	__SYSTEM.TYPE_CLASS.TYPE_ULINT:
	
	convertResult := TryConvert_TOD_TO_ULINT(in, _ULINT);
	IF convertResult THEN
		convertAddress := ADR(_ULINT);
	END_IF
	
	__SYSTEM.TYPE_CLASS.TYPE_REAL:
	
	convertResult := TryConvert_TOD_TO_REAL(in, _REAL);
	IF convertResult THEN
		convertAddress := ADR(_REAL);
	END_IF
	
	__SYSTEM.TYPE_CLASS.TYPE_LREAL:
	
	convertResult := TryConvert_TOD_TO_LREAL(in, _LREAL);
	IF convertResult THEN
		convertAddress := ADR(_LREAL);
	END_IF
	
	__SYSTEM.TYPE_CLASS.TYPE_TIME:
	
	convertResult := TryConvert_TOD_TO_TIME(in, _TIME);
	IF convertResult THEN
		convertAddress := ADR(_TIME);
	END_IF
	
	__SYSTEM.TYPE_CLASS.TYPE_TIMEOFDAY:
	
	convertResult := TryConvert_TOD_TO_TOD(in, _TOD);
	IF convertResult THEN
		convertAddress := ADR(_TOD);
	END_IF
	
	__SYSTEM.TYPE_CLASS.TYPE_DATE:
	
	convertResult := TryConvert_TOD_TO_DATE(in, _DATE);
	IF convertResult THEN
		convertAddress := ADR(_DATE);
	END_IF
	
	__SYSTEM.TYPE_CLASS.TYPE_DATEANDTIME:
	
	convertResult := TryConvert_TOD_TO_DT(in, _DT);
	IF convertResult THEN
		convertAddress := ADR(_DT);
	END_IF
	
	__SYSTEM.TYPE_CLASS.TYPE_STRING:
	
	convertResult := TryConvert_TOD_TO_STRING(in, _STRING);
	IF convertResult THEN
		convertAddress := ADR(_STRING);
	END_IF
	
END_CASE

IF convertResult THEN
	memcpy(out.pValue,convertAddress,DINT_TO_UDINT(out.diSize));
END_IF

TryConvert_TOD_TO_Destination := convertResult;

END_FUNCTION

// ---- mobject-datatypes/Primitive/_DT.TcPOU
{attribute 'linkalways'} 
{attribute 'no_explicit_call' := 'This FB is a CLASS and must be accessed using methods or properties'}
{attribute 'enable_dynamic_creation'}
FUNCTION_BLOCK _DT EXTENDS DatatypeBase implements I_DT
VAR
	localData : DT;
	activeData : REFERENCE TO DT REF= localData;
END_VAR

PROPERTY PUBLIC Address : PVOID
GET
Address := ADR(activeData);
END_GET
END_PROPERTY

METHOD PUBLIC ClearReference
VAR_INPUT
END_VAR
activeData REF= localData;
END_METHOD

METHOD PUBLIC Clone : I_Datatype
VAR
    pClone : POINTER TO _DT;
END_VAR
pClone := __NEW(_DT(InitialValue := Value));
Clone := pClone^;
END_METHOD

METHOD FB_init : BOOL
VAR_INPUT
	bInitRetains : BOOL; // if TRUE, the retain variables are initialized (warm start / cold start)
	bInCopyCode : BOOL;  // if TRUE, the instance afterwards gets moved WORDo the copy code (online change)
	InitialValue : DT;
END_VAR
localData := InitialValue;
END_METHOD

METHOD PUBLIC MakeReferenceTo
VAR_INPUT
	ReferenceTarget : REFERENCE TO DT;
END_VAR
activeData REF= ReferenceTarget;
END_METHOD

METHOD PUBLIC SerializeWith
VAR_INPUT
	Serializer : I_Serializer;
END_VAR
Serializer.AddDateTime(activeData);
END_METHOD

PROPERTY PUBLIC Size : UDINT
GET
Size := SIZEOF(activeData);
END_GET
END_PROPERTY

METHOD PUBLIC TryConvertTo : BOOL
VAR_INPUT
	Destination : ANY;
END_VAR
TryConvertTo := TryConvert_DT_To_Destination(activeData, Destination);
END_METHOD

METHOD PUBLIC TryConvertTo_ : BOOL
VAR_INPUT
	Destination : I_Datatype;
END_VAR
VAR
	resultofBitConversion : BOOL;
	destinationAs_BIT : I_BIT;
	destinationAs_BOOL : I_BOOL;
	destinationAs_BYTE : I_BYTE;
	destinationAs_DINT : I_DINT;
	destinationAs_DT : I_DT;
	destinationAs_DWORD : I_DWORD;
	destinationAs_INT : I_INT;
	destinationAs_LINT : I_LINT;
	destinationAs_LREAL : I_LREAL;
	destinationAs_LWORD : I_LWORD;
	destinationAs_REAL : I_REAL;
	destinationAs_SINT : I_SINT;
	destinationAs_STRING : I_STRING;
	destinationAs_TOD : I_TOD;
	destinationAs_UDINT : I_UDINT;
	destinationAs_UINT : I_UINT;
	destinationAs_ULINT : I_ULINT;
	destinationAs_USINT : I_USINT;
	destinationAs_WORD : I_WORD;
END_VAR
IF destination.TryResolveAs_BIT(destinationAs_BIT) AND_THEN TryConvert_DT_TO_BOOL(activeData, resultofBitConversion) THEN
	destinationAs_BIT.Value := resultOfBitConversion;
	TryConvertTo_ := TRUE;
	RETURN;
END_IF

IF destination.TryResolveAs_BOOL(destinationAs_BOOL) THEN
	TryConvertTo_ := TryConvert_DT_TO_BOOL(activeData, destinationAs_BOOL.Value);
	RETURN;
END_IF
		
IF destination.TryResolveAs_BYTE(destinationAs_BYTE) THEN
	TryConvertTo_ := TryConvert_DT_TO_BYTE(activeData, destinationAs_BYTE.Value);
	RETURN;
END_IF

IF destination.TryResolveAs_DINT(destinationAs_DINT) THEN
	TryConvertTo_ := TryConvert_DT_TO_DINT(activeData, destinationAs_DINT.Value);
	RETURN;
END_IF

IF destination.TryResolveAs_DT(destinationAs_DT) THEN
	TryConvertTo_ := TryConvert_DT_TO_DT(activeData, destinationAs_DT.Value);
	RETURN;
END_IF

IF destination.TryResolveAs_DWORD(destinationAs_DWORD) THEN
	TryConvertTo_ := TryConvert_DT_TO_DWORD(activeData, destinationAs_DWORD.Value);
	RETURN;
END_IF

IF destination.TryResolveAs_INT(destinationAs_INT) THEN
	TryConvertTo_ := TryConvert_DT_TO_INT(activeData, destinationAs_INT.Value);
	RETURN;
END_IF

IF destination.TryResolveAs_LINT(destinationAs_LINT) THEN
	TryConvertTo_ := TryConvert_DT_TO_LINT(activeData, destinationAs_LINT.Value);
	RETURN;
END_IF

IF destination.TryResolveAs_LREAL(destinationAs_LREAL) THEN
	TryConvertTo_ := TryConvert_DT_TO_LREAL(activeData, destinationAs_LREAL.Value);
	RETURN;
END_IF

IF destination.TryResolveAs_LWORD(destinationAs_LWORD) THEN
	TryConvertTo_ := TryConvert_DT_TO_LWORD(activeData, destinationAs_LWORD.Value);
	RETURN;
END_IF

IF destination.TryResolveAs_REAL(destinationAs_REAL) THEN
	TryConvertTo_ := TryConvert_DT_TO_REAL(activeData, destinationAs_REAL.Value);
	RETURN;
END_IF

IF destination.TryResolveAs_SINT(destinationAs_SINT) THEN
	TryConvertTo_ := TryConvert_DT_TO_SINT(activeData, destinationAs_SINT.Value);
	RETURN;
END_IF

IF destination.TryResolveAs_STRING(destinationAs_STRING) THEN
	TryConvertTo_ := TryConvert_DT_TO_STRING(activeData, destinationAs_STRING.Value);
	RETURN;
END_IF

IF destination.TryResolveAs_TOD(destinationAs_TOD) THEN
	TryConvertTo_ := TryConvert_DT_TO_TOD(activeData, destinationAs_TOD.Value);
	RETURN;
END_IF

IF destination.TryResolveAs_UDINT(destinationAs_UDINT) THEN
	TryConvertTo_ := TryConvert_DT_TO_UDINT(activeData, destinationAs_UDINT.Value);
	RETURN;
END_IF

IF destination.TryResolveAs_UINT(destinationAs_UINT) THEN
	TryConvertTo_ := TryConvert_DT_TO_UINT(activeData, destinationAs_UINT.Value);
	RETURN;
END_IF

IF destination.TryResolveAs_ULINT(destinationAs_ULINT) THEN
	TryConvertTo_ := TryConvert_DT_TO_ULINT(activeData, destinationAs_ULINT.Value);
	RETURN;
END_IF

IF destination.TryResolveAs_USINT(destinationAs_USINT) THEN
	TryConvertTo_ := TryConvert_DT_TO_USINT(activeData, destinationAs_USINT.Value);
	RETURN;
END_IF

IF destination.TryResolveAs_WORD(destinationAs_WORD) THEN
	TryConvertTo_ := TryConvert_DT_TO_WORD(activeData, destinationAs_WORD.Value);
	RETURN;
END_IF
END_METHOD

METHOD TryDeserializeFrom : BOOL
VAR_INPUT
	Deserializer : I_Deserializer;
	Feedback : I_DeserializerFeedback;
END_VAR
TryDeserializeFrom := Deserializer.TryGetDateTime(activeData, Feedback);
END_METHOD

METHOD TryMakeReferenceTo : BOOL
VAR_INPUT
	Target : I_Datatype;
END_VAR
VAR
	pTargetData : POINTER TO DT;
END_VAR
IF NOT IsEquivalentTo(Target) THEN
	RETURN;
END_IF

pTargetData := Target.Address;
activeData REF= pTargetData^;
TryMakeReferenceTo := TRUE;
END_METHOD

METHOD PUBLIC TryResolveAs_DT : BOOL
VAR_INPUT
	Destination : REFERENCE TO I_DT;
END_VAR
Destination := THIS^;
TryResolveAs_DT := TRUE;
END_METHOD

PROPERTY PUBLIC TypeName : T_MAXSTRING
GET
TypeName := 'DT';
END_GET
END_PROPERTY

{warning disable C5410}
PROPERTY PUBLIC Value : REFERENCE TO DT
{warning restore C5410}
GET
Value REF= activeData;
END_GET
END_PROPERTY

END_FUNCTION_BLOCK

// ---- mobject-converters/Converters/DT_TO_/TryConvert_DT_TO_BOOL.TcPOU
FUNCTION TryConvert_DT_TO_BOOL : BOOL
VAR_INPUT
	in : DT;
	out : REFERENCE TO BOOL;
END_VAR

out := DT_TO_BOOL(in);
TryConvert_DT_TO_BOOL := TRUE;

END_FUNCTION

// ---- mobject-converters/Converters/DT_TO_/TryConvert_DT_TO_BYTE.TcPOU
FUNCTION TryConvert_DT_TO_BYTE : BOOL
VAR_INPUT
	in : DT;
	out : REFERENCE TO BYTE;
END_VAR

IF in > DatatypeLimits.MAX_VALUE_OF_DT_WHICH_CAN_BE_HELD_IN_A_BYTE THEN
	RETURN;
END_IF

out := DT_TO_BYTE(in);
TryConvert_DT_TO_BYTE := TRUE;

END_FUNCTION

// ---- mobject-converters/Converters/DT_TO_/TryConvert_DT_TO_DINT.TcPOU
FUNCTION TryConvert_DT_TO_DINT : BOOL
VAR_INPUT
	in : DT;
	out : REFERENCE TO DINT;
END_VAR

IF in > DatatypeLimits.MAX_VALUE_OF_DT_WHICH_CAN_BE_HELD_IN_A_DINT THEN
	RETURN;
END_IF

out := DT_TO_DINT(in);
TryConvert_DT_TO_DINT := TRUE;

END_FUNCTION

// ---- mobject-converters/Converters/DT_TO_/TryConvert_DT_TO_DT.TcPOU
FUNCTION TryConvert_DT_TO_DT : BOOL
VAR_INPUT
	in : DT;
	out : REFERENCE TO DT;
END_VAR

out := in;
TryConvert_DT_TO_DT := TRUE;

END_FUNCTION

// ---- mobject-converters/Converters/DT_TO_/TryConvert_DT_TO_DWORD.TcPOU
FUNCTION TryConvert_DT_TO_DWORD : BOOL
VAR_INPUT
	in : DT;
	out : REFERENCE TO DWORD;
END_VAR

out := DT_TO_DWORD(in);
TryConvert_DT_TO_DWORD := TRUE;

END_FUNCTION

// ---- mobject-converters/Converters/DT_TO_/TryConvert_DT_TO_LINT.TcPOU
FUNCTION TryConvert_DT_TO_LINT : BOOL
VAR_INPUT
	in : DT;
	out : REFERENCE TO LINT;
END_VAR

out := DT_TO_LINT(in);
TryConvert_DT_TO_LINT := TRUE;

END_FUNCTION

// ---- mobject-converters/Converters/DT_TO_/TryConvert_DT_TO_LWORD.TcPOU
FUNCTION TryConvert_DT_TO_LWORD : BOOL
VAR_INPUT
	in : DT;
	out : REFERENCE TO LWORD;
END_VAR

out := DT_TO_LWORD(in);
TryConvert_DT_TO_LWORD := TRUE;

END_FUNCTION

// ---- mobject-converters/Converters/DT_TO_/TryConvert_DT_TO_REAL.TcPOU
FUNCTION TryConvert_DT_TO_REAL : BOOL
VAR_INPUT
	in : DT;
	out : REFERENCE TO REAL;
END_VAR

out := DT_TO_REAL(in);
TryConvert_DT_TO_REAL := TRUE;

END_FUNCTION

// ---- mobject-converters/Converters/DT_TO_/TryConvert_DT_TO_TOD.TcPOU
FUNCTION TryConvert_DT_TO_TOD : BOOL
VAR_INPUT
	in : DT;
	out : REFERENCE TO TOD;
END_VAR

IF in > DatatypeLimits.MAX_VALUE_OF_DT_WHICH_CAN_BE_HELD_IN_A_TOD THEN
	RETURN;
END_IF

out := DT_TO_TOD(in);
TryConvert_DT_TO_TOD := TRUE;

END_FUNCTION

// ---- mobject-converters/Converters/DT_TO_/TryConvert_DT_TO_UINT.TcPOU
FUNCTION TryConvert_DT_TO_UINT : BOOL
VAR_INPUT
	in : DT;
	out : REFERENCE TO UINT;
END_VAR

IF in > DatatypeLimits.MAX_VALUE_OF_DT_WHICH_CAN_BE_HELD_IN_A_UINT THEN
	RETURN;
END_IF

out := DT_TO_UINT(in);
TryConvert_DT_TO_UINT := TRUE;

END_FUNCTION

// ---- mobject-converters/Converters/DT_TO_/TryConvert_DT_TO_ULINT.TcPOU
FUNCTION TryConvert_DT_TO_ULINT : BOOL
VAR_INPUT
	in : DT;
	out : REFERENCE TO ULINT;
END_VAR

out := DT_TO_ULINT(in);
TryConvert_DT_TO_ULINT := TRUE;

END_FUNCTION

// ---- mobject-datatypes/Primitive/_STRING.TcPOU
{attribute 'linkalways'} 
{attribute 'no_explicit_call' := 'This FB is a CLASS and must be accessed using methods or properties'}
{attribute 'enable_dynamic_creation'}
FUNCTION_BLOCK _STRING EXTENDS DatatypeBase implements I_STRING
VAR
	localData : T_MaxString;
	activeData : REFERENCE TO T_MaxString REF= localData;
END_VAR

PROPERTY PUBLIC Address : PVOID
GET
Address := ADR(activeData);
END_GET
END_PROPERTY

METHOD PUBLIC ClearReference
VAR_INPUT
END_VAR
activeData REF= localData;
END_METHOD

METHOD PUBLIC Clone : I_Datatype
VAR
    pClone : POINTER TO _STRING;
END_VAR
pClone := __NEW(_STRING(InitialValue := Value));
Clone := pClone^;
END_METHOD

METHOD FB_init : BOOL
VAR_INPUT
	bInitRetains : BOOL; // if TRUE, the retain variables are initialized (warm start / cold start)
	bInCopyCode : BOOL;  // if TRUE, the instance afterwards gets moved WORDo the copy code (online change)
	InitialValue : T_MaxString;
END_VAR
localData := InitialValue;
END_METHOD

PROPERTY PUBLIC Length : INT
GET
Length := len(activeData);
END_GET
END_PROPERTY

METHOD PUBLIC MakeReferenceTo
VAR_INPUT
	ReferenceTarget : REFERENCE TO T_MaxString;
END_VAR
activeData REF= ReferenceTarget;
END_METHOD

METHOD PUBLIC SerializeWith
VAR_INPUT
	Serializer : I_Serializer;
END_VAR
Serializer.AddString(activeData);
END_METHOD

PROPERTY PUBLIC Size : UDINT
GET
Size := SIZEOF(activeData);
END_GET
END_PROPERTY

METHOD PUBLIC TryConvertTo : BOOL
VAR_INPUT
	Destination : ANY;
END_VAR
TryConvertTo := TryConvert_STRING_TO_Destination(activeData, Destination);
END_METHOD

METHOD PUBLIC TryConvertTo_ : BOOL
VAR_INPUT
	Destination : I_Datatype;
END_VAR
VAR
	resultofBitConversion : BOOL;
	destinationAs_BIT : I_BIT;
	destinationAs_BOOL : I_BOOL;
	destinationAs_BYTE : I_BYTE;
	destinationAs_DINT : I_DINT;
	destinationAs_DT : I_DT;
	destinationAs_DWORD : I_DWORD;
	destinationAs_INT : I_INT;
	destinationAs_LINT : I_LINT;
	destinationAs_LREAL : I_LREAL;
	destinationAs_LWORD : I_LWORD;
	destinationAs_REAL : I_REAL;
	destinationAs_SINT : I_SINT;
	destinationAs_STRING : I_STRING;
	destinationAs_TOD : I_TOD;
	destinationAs_UDINT : I_UDINT;
	destinationAs_UINT : I_UINT;
	destinationAs_ULINT : I_ULINT;
	destinationAs_USINT : I_USINT;
	destinationAs_WORD : I_WORD;
END_VAR
IF destination.TryResolveAs_BIT(destinationAs_BIT) AND_THEN TryConvert_STRING_TO_BOOL(activeData, resultofBitConversion) THEN
	destinationAs_BIT.Value := resultOfBitConversion;
	TryConvertTo_ := TRUE;
	RETURN;
END_IF

IF destination.TryResolveAs_BOOL(destinationAs_BOOL) THEN
	TryConvertTo_ := TryConvert_STRING_TO_BOOL(activeData, destinationAs_BOOL.Value);
	RETURN;
END_IF
		
IF destination.TryResolveAs_BYTE(destinationAs_BYTE) THEN
	TryConvertTo_ := TryConvert_STRING_TO_BYTE(activeData, destinationAs_BYTE.Value);
	RETURN;
END_IF

IF destination.TryResolveAs_DINT(destinationAs_DINT) THEN
	TryConvertTo_ := TryConvert_STRING_TO_DINT(activeData, destinationAs_DINT.Value);
	RETURN;
END_IF

IF destination.TryResolveAs_DT(destinationAs_DT) THEN
	TryConvertTo_ := TryConvert_STRING_TO_DT(activeData, destinationAs_DT.Value);
	RETURN;
END_IF

IF destination.TryResolveAs_DWORD(destinationAs_DWORD) THEN
	TryConvertTo_ := TryConvert_STRING_TO_DWORD(activeData, destinationAs_DWORD.Value);
	RETURN;
END_IF

IF destination.TryResolveAs_INT(destinationAs_INT) THEN
	TryConvertTo_ := TryConvert_STRING_TO_INT(activeData, destinationAs_INT.Value);
	RETURN;
END_IF

IF destination.TryResolveAs_LINT(destinationAs_LINT) THEN
	TryConvertTo_ := TryConvert_STRING_TO_LINT(activeData, destinationAs_LINT.Value);
	RETURN;
END_IF

IF destination.TryResolveAs_LREAL(destinationAs_LREAL) THEN
	TryConvertTo_ := TryConvert_STRING_TO_LREAL(activeData, destinationAs_LREAL.Value);
	RETURN;
END_IF

IF destination.TryResolveAs_LWORD(destinationAs_LWORD) THEN
	TryConvertTo_ := TryConvert_STRING_TO_LWORD(activeData, destinationAs_LWORD.Value);
	RETURN;
END_IF

IF destination.TryResolveAs_REAL(destinationAs_REAL) THEN
	TryConvertTo_ := TryConvert_STRING_TO_REAL(activeData, destinationAs_REAL.Value);
	RETURN;
END_IF

IF destination.TryResolveAs_SINT(destinationAs_SINT) THEN
	TryConvertTo_ := TryConvert_STRING_TO_SINT(activeData, destinationAs_SINT.Value);
	RETURN;
END_IF

IF destination.TryResolveAs_STRING(destinationAs_STRING) THEN
	TryConvertTo_ := TryConvert_STRING_TO_STRING(activeData, destinationAs_STRING.Value);
	RETURN;
END_IF

IF destination.TryResolveAs_TOD(destinationAs_TOD) THEN
	TryConvertTo_ := TryConvert_STRING_TO_TOD(activeData, destinationAs_TOD.Value);
	RETURN;
END_IF

IF destination.TryResolveAs_UDINT(destinationAs_UDINT) THEN
	TryConvertTo_ := TryConvert_STRING_TO_UDINT(activeData, destinationAs_UDINT.Value);
	RETURN;
END_IF

IF destination.TryResolveAs_UINT(destinationAs_UINT) THEN
	TryConvertTo_ := TryConvert_STRING_TO_UINT(activeData, destinationAs_UINT.Value);
	RETURN;
END_IF

IF destination.TryResolveAs_ULINT(destinationAs_ULINT) THEN
	TryConvertTo_ := TryConvert_STRING_TO_ULINT(activeData, destinationAs_ULINT.Value);
	RETURN;
END_IF

IF destination.TryResolveAs_USINT(destinationAs_USINT) THEN
	TryConvertTo_ := TryConvert_STRING_TO_USINT(activeData, destinationAs_USINT.Value);
	RETURN;
END_IF

IF destination.TryResolveAs_WORD(destinationAs_WORD) THEN
	TryConvertTo_ := TryConvert_STRING_TO_WORD(activeData, destinationAs_WORD.Value);
	RETURN;
END_IF
END_METHOD

METHOD TryDeserializeFrom : BOOL
VAR_INPUT
	Deserializer : I_Deserializer;
	Feedback : I_DeserializerFeedback;
END_VAR
TryDeserializeFrom := Deserializer.TryGetString(activeData, Feedback);
END_METHOD

METHOD TryMakeReferenceTo : BOOL
VAR_INPUT
	Target : I_Datatype;
END_VAR
VAR
	pTargetData : POINTER TO T_MaxString;
END_VAR
IF NOT IsEquivalentTo(Target) THEN
	RETURN;
END_IF

pTargetData := Target.Address;
activeData REF= pTargetData^;
TryMakeReferenceTo := TRUE;
END_METHOD

METHOD PUBLIC TryResolveAs_STRING : BOOL
VAR_INPUT
	Destination : REFERENCE TO I_STRING;
END_VAR
Destination := THIS^;
TryResolveAs_STRING := TRUE;
END_METHOD

PROPERTY PUBLIC TypeName : T_MAXSTRING
GET
TypeName := 'STRING';
END_GET
END_PROPERTY

{warning disable C5410}
PROPERTY PUBLIC Value : REFERENCE TO T_MaxString
{warning restore C5410}
GET
Value REF= activeData;
END_GET
END_PROPERTY

END_FUNCTION_BLOCK

// ---- mobject-converters/Converters/STRING_TO_/TryConvert_STRING_TO_Destination.TcPOU
FUNCTION TryConvert_STRING_TO_Destination : BOOL
VAR_INPUT
	in : STRING;
	out : ANY;
END_VAR
VAR
	convertResult : BOOL := FALSE;
	convertAddress : PVOID;
	_BOOL : BOOL;
	_BYTE : BYTE;
	_WORD : WORD;
	_DWORD : DWORD;
	_LWORD : LWORD;
	_SINT : SINT;
	_INT : INT;
	_DINT : DINT;
	_LINT : LINT;
	_USINT : USINT;
	_UINT : UINT;
	_UDINT : UDINT;
	_ULINT : ULINT;
	_REAL : REAL;
	_LREAL : LREAL;
	_TIME : TIME;
	_TOD : TOD;
	_DATE : DATE;
	_DT : DT;
	_STRING : STRING;
END_VAR

CASE out.TypeClass OF
	__SYSTEM.TYPE_CLASS.TYPE_BOOL:
	
	convertResult := TryConvert_STRING_TO_BOOL(in, _BOOL);
	IF convertResult THEN
		convertAddress := ADR(_BOOL);
	END_IF
	
	__SYSTEM.TYPE_CLASS.TYPE_BYTE:
	
	convertResult := TryConvert_STRING_TO_BYTE(in, _BYTE);
	IF convertResult THEN
		convertAddress := ADR(_BYTE);
	END_IF
	
	__SYSTEM.TYPE_CLASS.TYPE_WORD:
	
	convertResult := TryConvert_STRING_TO_WORD(in, _WORD);
	IF convertResult THEN
		convertAddress := ADR(_WORD);
	END_IF
	
	__SYSTEM.TYPE_CLASS.TYPE_DWORD:
	
	convertResult := TryConvert_STRING_TO_DWORD(in, _DWORD);
	IF convertResult THEN
		convertAddress := ADR(_DWORD);
	END_IF
	
	__SYSTEM.TYPE_CLASS.TYPE_LWORD:
	
	convertResult := TryConvert_STRING_TO_LWORD(in, _LWORD);
	IF convertResult THEN
		convertAddress := ADR(_LWORD);
	END_IF
	
	__SYSTEM.TYPE_CLASS.TYPE_SINT:
	
	convertResult := TryConvert_STRING_TO_SINT(in, _SINT);
	IF convertResult THEN
		convertAddress := ADR(_SINT);
	END_IF
	
	__SYSTEM.TYPE_CLASS.TYPE_INT:
	
	convertResult := TryConvert_STRING_TO_INT(in, _INT);
	IF convertResult THEN
		convertAddress := ADR(_INT);
	END_IF
	
	__SYSTEM.TYPE_CLASS.TYPE_DINT:
	
	convertResult := TryConvert_STRING_TO_DINT(in, _DINT);
	IF convertResult THEN
		convertAddress := ADR(_DINT);
	END_IF
	
	__SYSTEM.TYPE_CLASS.TYPE_LINT:
	
	convertResult := TryConvert_STRING_TO_LINT(in, _LINT);
	IF convertResult THEN
		convertAddress := ADR(_LINT);
	END_IF
	
	__SYSTEM.TYPE_CLASS.TYPE_USINT:
	
	convertResult := TryConvert_STRING_TO_USINT(in, _USINT);
	IF convertResult THEN
		convertAddress := ADR(_USINT);
	END_IF
	
	__SYSTEM.TYPE_CLASS.TYPE_UINT:
	
	convertResult := TryConvert_STRING_TO_UINT(in, _UINT);
	IF convertResult THEN
		convertAddress := ADR(_UINT);
	END_IF
	
	__SYSTEM.TYPE_CLASS.TYPE_UDINT:
	
	convertResult := TryConvert_STRING_TO_UDINT(in, _UDINT);
	IF convertResult THEN
		convertAddress := ADR(_UDINT);
	END_IF
	
	__SYSTEM.TYPE_CLASS.TYPE_ULINT:
	
	convertResult := TryConvert_STRING_TO_ULINT(in, _ULINT);
	IF convertResult THEN
		convertAddress := ADR(_ULINT);
	END_IF
	
	__SYSTEM.TYPE_CLASS.TYPE_REAL:
	
	convertResult := TryConvert_STRING_TO_REAL(in, _REAL);
	IF convertResult THEN
		convertAddress := ADR(_REAL);
	END_IF
	
	__SYSTEM.TYPE_CLASS.TYPE_LREAL:
	
	convertResult := TryConvert_STRING_TO_LREAL(in, _LREAL);
	IF convertResult THEN
		convertAddress := ADR(_LREAL);
	END_IF
	
	__SYSTEM.TYPE_CLASS.TYPE_TIME:
	
	convertResult := TryConvert_STRING_TO_TIME(in, _TIME);
	IF convertResult THEN
		convertAddress := ADR(_TIME);
	END_IF
	
	__SYSTEM.TYPE_CLASS.TYPE_TIMEOFDAY:
	
	convertResult := TryConvert_STRING_TO_TOD(in, _TOD);
	IF convertResult THEN
		convertAddress := ADR(_TOD);
	END_IF
	
	__SYSTEM.TYPE_CLASS.TYPE_DATE:
	
	convertResult := TryConvert_STRING_TO_DATE(in, _DATE);
	IF convertResult THEN
		convertAddress := ADR(_DATE);
	END_IF
	
	__SYSTEM.TYPE_CLASS.TYPE_DATEANDTIME:
	
	convertResult := TryConvert_STRING_TO_DT(in, _DT);
	IF convertResult THEN
		convertAddress := ADR(_DT);
	END_IF
	
	__SYSTEM.TYPE_CLASS.TYPE_STRING:
	
	convertResult := TryConvert_STRING_TO_STRING(in, _STRING);
	IF convertResult THEN
		convertAddress := ADR(_STRING);
	END_IF
	
END_CASE

IF convertResult THEN
	memcpy(out.pValue,convertAddress,DINT_TO_UDINT(out.diSize));
END_IF

TryConvert_STRING_TO_Destination := convertResult;

END_FUNCTION

// ---- mobject-converters/Converters/STRING_TO_/TryConvert_STRING_TO_BYTE.TcPOU
FUNCTION TryConvert_STRING_TO_BYTE : BOOL
VAR_INPUT
	in : STRING;
	out : REFERENCE TO BYTE;
END_VAR

IF in <> BYTE_TO_STRING(STRING_TO_BYTE(in)) THEN
	RETURN;
END_IF

out := STRING_TO_BYTE(in);
TryConvert_STRING_TO_BYTE := TRUE;

END_FUNCTION

// ---- mobject-converters/Converters/STRING_TO_/TryConvert_STRING_TO_WORD.TcPOU
FUNCTION TryConvert_STRING_TO_WORD : BOOL
VAR_INPUT
	in : STRING;
	out : REFERENCE TO WORD;
END_VAR

IF in <> WORD_TO_STRING(STRING_TO_WORD(in)) THEN
	RETURN;
END_IF

out := STRING_TO_WORD(in);
TryConvert_STRING_TO_WORD := TRUE;

END_FUNCTION

// ---- mobject-converters/Converters/STRING_TO_/TryConvert_STRING_TO_DWORD.TcPOU
FUNCTION TryConvert_STRING_TO_DWORD : BOOL
VAR_INPUT
	in : STRING;
	out : REFERENCE TO DWORD;
END_VAR

IF in <> DWORD_TO_STRING(STRING_TO_DWORD(in)) THEN
	RETURN;
END_IF

out := STRING_TO_DWORD(in);
TryConvert_STRING_TO_DWORD := TRUE;

END_FUNCTION

// ---- mobject-converters/Converters/STRING_TO_/TryConvert_STRING_TO_SINT.TcPOU
FUNCTION TryConvert_STRING_TO_SINT : BOOL
VAR_INPUT
	in : STRING;
	out : REFERENCE TO SINT;
END_VAR

IF in <> SINT_TO_STRING(STRING_TO_SINT(in)) THEN
	RETURN;
END_IF

out := STRING_TO_SINT(in);
TryConvert_STRING_TO_SINT := TRUE;

END_FUNCTION

// ---- mobject-converters/Converters/STRING_TO_/TryConvert_STRING_TO_DINT.TcPOU
FUNCTION TryConvert_STRING_TO_DINT : BOOL
VAR_INPUT
	in : STRING;
	out : REFERENCE TO DINT;
END_VAR

IF in <> DINT_TO_STRING(STRING_TO_DINT(in)) THEN
	RETURN;
END_IF

out := STRING_TO_DINT(in);
TryConvert_STRING_TO_DINT := TRUE;

END_FUNCTION

// ---- mobject-converters/Converters/STRING_TO_/TryConvert_STRING_TO_USINT.TcPOU
FUNCTION TryConvert_STRING_TO_USINT : BOOL
VAR_INPUT
	in : STRING;
	out : REFERENCE TO USINT;
END_VAR

IF in <> USINT_TO_STRING(STRING_TO_USINT(in)) THEN
	RETURN;
END_IF

out := STRING_TO_USINT(in);
TryConvert_STRING_TO_USINT := TRUE;

END_FUNCTION

// ---- mobject-converters/Converters/STRING_TO_/TryConvert_STRING_TO_UINT.TcPOU
FUNCTION TryConvert_STRING_TO_UINT : BOOL
VAR_INPUT
	in : STRING;
	out : REFERENCE TO UINT;
END_VAR

IF in <> UINT_TO_STRING(STRING_TO_UINT(in)) THEN
	RETURN;
END_IF

out := STRING_TO_UINT(in);
TryConvert_STRING_TO_UINT := TRUE;

END_FUNCTION

// ---- mobject-converters/Converters/STRING_TO_/TryConvert_STRING_TO_ULINT.TcPOU
FUNCTION TryConvert_STRING_TO_ULINT : BOOL
VAR_INPUT
	in : STRING;
	out : REFERENCE TO ULINT;
END_VAR

IF in <> ULINT_TO_STRING(STRING_TO_ULINT(in)) THEN
	RETURN;
END_IF

out := STRING_TO_ULINT(in);
TryConvert_STRING_TO_ULINT := TRUE;

END_FUNCTION

// ---- mobject-converters/Converters/STRING_TO_/TryConvert_STRING_TO_REAL.TcPOU
FUNCTION TryConvert_STRING_TO_REAL : BOOL
VAR_INPUT
	in : STRING;
	out : REFERENCE TO REAL;
END_VAR

IF in <> REAL_TO_STRING(STRING_TO_REAL(in)) THEN
	RETURN;
END_IF

out := STRING_TO_REAL(in);
TryConvert_STRING_TO_REAL := TRUE;

END_FUNCTION

// ---- mobject-converters/Converters/STRING_TO_/TryConvert_STRING_TO_LREAL.TcPOU
FUNCTION TryConvert_STRING_TO_LREAL : BOOL
VAR_INPUT
	in : STRING;
	out : REFERENCE TO LREAL;
END_VAR

IF in <> LREAL_TO_STRING(STRING_TO_LREAL(in)) THEN
	RETURN;
END_IF

out := STRING_TO_LREAL(in);
TryConvert_STRING_TO_LREAL := TRUE;

END_FUNCTION

// ---- mobject-converters/Converters/STRING_TO_/TryConvert_STRING_TO_TOD.TcPOU
FUNCTION TryConvert_STRING_TO_TOD : BOOL
VAR_INPUT
	in : STRING;
	out : REFERENCE TO TOD;
END_VAR

IF in <> TOD_TO_STRING(STRING_TO_TOD(in)) THEN
	RETURN;
END_IF

out := STRING_TO_TOD(in);
TryConvert_STRING_TO_TOD := TRUE;

END_FUNCTION

// ---- mobject-converters/Converters/STRING_TO_/TryConvert_STRING_TO_DATE.TcPOU
FUNCTION TryConvert_STRING_TO_DATE : BOOL
VAR_INPUT
	in : STRING;
	out : REFERENCE TO DATE;
END_VAR

IF in <> DATE_TO_STRING(STRING_TO_DATE(in)) THEN
	RETURN;
END_IF

out := STRING_TO_DATE(in);
TryConvert_STRING_TO_DATE := TRUE;

END_FUNCTION

// ---- mobject-converters/Converters/STRING_TO_/TryConvert_STRING_TO_STRING.TcPOU
FUNCTION TryConvert_STRING_TO_STRING : BOOL
VAR_INPUT
	in : STRING;
	out : REFERENCE TO STRING;
END_VAR

out := in;
TryConvert_STRING_TO_STRING := TRUE;

END_FUNCTION

// ---- mobject-converters/Converters/TOD_TO_/TryConvert_TOD_TO_BOOL.TcPOU
FUNCTION TryConvert_TOD_TO_BOOL : BOOL
VAR_INPUT
	in : TOD;
	out : REFERENCE TO BOOL;
END_VAR

out := TOD_TO_BOOL(in);
TryConvert_TOD_TO_BOOL := TRUE;

END_FUNCTION

// ---- mobject-converters/Converters/TOD_TO_/TryConvert_TOD_TO_BYTE.TcPOU
FUNCTION TryConvert_TOD_TO_BYTE : BOOL
VAR_INPUT
	in : TOD;
	out : REFERENCE TO BYTE;
END_VAR

IF in > DatatypeLimits.MAX_VALUE_OF_TOD_WHICH_CAN_BE_HELD_IN_A_BYTE THEN
	RETURN;
END_IF

out := TOD_TO_BYTE(in);
TryConvert_TOD_TO_BYTE := TRUE;

END_FUNCTION

// ---- mobject-converters/Converters/TOD_TO_/TryConvert_TOD_TO_WORD.TcPOU
FUNCTION TryConvert_TOD_TO_WORD : BOOL
VAR_INPUT
	in : TOD;
	out : REFERENCE TO WORD;
END_VAR

IF in > DatatypeLimits.MAX_VALUE_OF_TOD_WHICH_CAN_BE_HELD_IN_A_WORD THEN
	RETURN;
END_IF

out := TOD_TO_WORD(in);
TryConvert_TOD_TO_WORD := TRUE;

END_FUNCTION

// ---- mobject-converters/Converters/TOD_TO_/TryConvert_TOD_TO_INT.TcPOU
FUNCTION TryConvert_TOD_TO_INT : BOOL
VAR_INPUT
	in : TOD;
	out : REFERENCE TO INT;
END_VAR

IF in > DatatypeLimits.MAX_VALUE_OF_TOD_WHICH_CAN_BE_HELD_IN_A_INT THEN
	RETURN;
END_IF

out := TOD_TO_INT(in);
TryConvert_TOD_TO_INT := TRUE;

END_FUNCTION

// ---- mobject-converters/Converters/TOD_TO_/TryConvert_TOD_TO_LINT.TcPOU
FUNCTION TryConvert_TOD_TO_LINT : BOOL
VAR_INPUT
	in : TOD;
	out : REFERENCE TO LINT;
END_VAR

out := TOD_TO_LINT(in);
TryConvert_TOD_TO_LINT := TRUE;

END_FUNCTION

// ---- mobject-converters/Converters/TOD_TO_/TryConvert_TOD_TO_USINT.TcPOU
FUNCTION TryConvert_TOD_TO_USINT : BOOL
VAR_INPUT
	in : TOD;
	out : REFERENCE TO USINT;
END_VAR

IF in > DatatypeLimits.MAX_VALUE_OF_TOD_WHICH_CAN_BE_HELD_IN_A_USINT THEN
	RETURN;
END_IF

out := TOD_TO_USINT(in);
TryConvert_TOD_TO_USINT := TRUE;

END_FUNCTION

// ---- mobject-converters/Converters/TOD_TO_/TryConvert_TOD_TO_REAL.TcPOU
FUNCTION TryConvert_TOD_TO_REAL : BOOL
VAR_INPUT
	in : TOD;
	out : REFERENCE TO REAL;
END_VAR

out := TOD_TO_REAL(in);
TryConvert_TOD_TO_REAL := TRUE;

END_FUNCTION

// ---- mobject-converters/Converters/TOD_TO_/TryConvert_TOD_TO_TIME.TcPOU
FUNCTION TryConvert_TOD_TO_TIME : BOOL
VAR_INPUT
	in : TOD;
	out : REFERENCE TO TIME;
END_VAR

out := TOD_TO_TIME(in);
TryConvert_TOD_TO_TIME := TRUE;

END_FUNCTION

// ---- mobject-converters/Converters/ULINT_TO_/TryConvert_ULINT_TO_BYTE.TcPOU
FUNCTION TryConvert_ULINT_TO_BYTE : BOOL
VAR_INPUT
	in : ULINT;
	out : REFERENCE TO BYTE;
END_VAR

IF in > DatatypeLimits.MAX_VALUE_OF_ULINT_WHICH_CAN_BE_HELD_IN_A_BYTE THEN
	RETURN;
END_IF

out := ULINT_TO_BYTE(in);
TryConvert_ULINT_TO_BYTE := TRUE;

END_FUNCTION

// ---- mobject-converters/Converters/ULINT_TO_/TryConvert_ULINT_TO_WORD.TcPOU
FUNCTION TryConvert_ULINT_TO_WORD : BOOL
VAR_INPUT
	in : ULINT;
	out : REFERENCE TO WORD;
END_VAR

IF in > DatatypeLimits.MAX_VALUE_OF_ULINT_WHICH_CAN_BE_HELD_IN_A_WORD THEN
	RETURN;
END_IF

out := ULINT_TO_WORD(in);
TryConvert_ULINT_TO_WORD := TRUE;

END_FUNCTION

// ---- mobject-converters/Converters/ULINT_TO_/TryConvert_ULINT_TO_DWORD.TcPOU
FUNCTION TryConvert_ULINT_TO_DWORD : BOOL
VAR_INPUT
	in : ULINT;
	out : REFERENCE TO DWORD;
END_VAR

IF in > DatatypeLimits.MAX_VALUE_OF_ULINT_WHICH_CAN_BE_HELD_IN_A_DWORD THEN
	RETURN;
END_IF

out := ULINT_TO_DWORD(in);
TryConvert_ULINT_TO_DWORD := TRUE;

END_FUNCTION

// ---- mobject-converters/Converters/ULINT_TO_/TryConvert_ULINT_TO_INT.TcPOU
FUNCTION TryConvert_ULINT_TO_INT : BOOL
VAR_INPUT
	in : ULINT;
	out : REFERENCE TO INT;
END_VAR

IF in > DatatypeLimits.MAX_VALUE_OF_ULINT_WHICH_CAN_BE_HELD_IN_A_INT THEN
	RETURN;
END_IF

out := ULINT_TO_INT(in);
TryConvert_ULINT_TO_INT := TRUE;

END_FUNCTION

// ---- mobject-converters/Converters/ULINT_TO_/TryConvert_ULINT_TO_LINT.TcPOU
FUNCTION TryConvert_ULINT_TO_LINT : BOOL
VAR_INPUT
	in : ULINT;
	out : REFERENCE TO LINT;
END_VAR

IF in > DatatypeLimits.MAX_VALUE_OF_ULINT_WHICH_CAN_BE_HELD_IN_A_LINT THEN
	RETURN;
END_IF

out := ULINT_TO_LINT(in);
TryConvert_ULINT_TO_LINT := TRUE;

END_FUNCTION

// ---- mobject-converters/Converters/ULINT_TO_/TryConvert_ULINT_TO_UINT.TcPOU
FUNCTION TryConvert_ULINT_TO_UINT : BOOL
VAR_INPUT
	in : ULINT;
	out : REFERENCE TO UINT;
END_VAR

IF in > DatatypeLimits.MAX_VALUE_OF_ULINT_WHICH_CAN_BE_HELD_IN_A_UINT THEN
	RETURN;
END_IF

out := ULINT_TO_UINT(in);
TryConvert_ULINT_TO_UINT := TRUE;

END_FUNCTION

// ---- mobject-converters/Converters/ULINT_TO_/TryConvert_ULINT_TO_ULINT.TcPOU
FUNCTION TryConvert_ULINT_TO_ULINT : BOOL
VAR_INPUT
	in : ULINT;
	out : REFERENCE TO ULINT;
END_VAR

out := in;
TryConvert_ULINT_TO_ULINT := TRUE;

END_FUNCTION

// ---- mobject-converters/Converters/ULINT_TO_/TryConvert_ULINT_TO_REAL.TcPOU
FUNCTION TryConvert_ULINT_TO_REAL : BOOL
VAR_INPUT
	in : ULINT;
	out : REFERENCE TO REAL;
END_VAR

out := ULINT_TO_REAL(in);
TryConvert_ULINT_TO_REAL := TRUE;

END_FUNCTION

// ---- mobject-converters/Converters/ULINT_TO_/TryConvert_ULINT_TO_LREAL.TcPOU
FUNCTION TryConvert_ULINT_TO_LREAL : BOOL
VAR_INPUT
	in : ULINT;
	out : REFERENCE TO LREAL;
END_VAR

out := ULINT_TO_LREAL(in);
TryConvert_ULINT_TO_LREAL := TRUE;

END_FUNCTION

// ---- mobject-converters/Converters/ULINT_TO_/TryConvert_ULINT_TO_TIME.TcPOU
FUNCTION TryConvert_ULINT_TO_TIME : BOOL
VAR_INPUT
	in : ULINT;
	out : REFERENCE TO TIME;
END_VAR

IF in > DatatypeLimits.MAX_VALUE_OF_ULINT_WHICH_CAN_BE_HELD_IN_A_TIME THEN
	RETURN;
END_IF

out := ULINT_TO_TIME(in);
TryConvert_ULINT_TO_TIME := TRUE;

END_FUNCTION

// ---- mobject-converters/Converters/ULINT_TO_/TryConvert_ULINT_TO_TOD.TcPOU
FUNCTION TryConvert_ULINT_TO_TOD : BOOL
VAR_INPUT
	in : ULINT;
	out : REFERENCE TO TOD;
END_VAR

IF in > DatatypeLimits.MAX_VALUE_OF_ULINT_WHICH_CAN_BE_HELD_IN_A_TOD THEN
	RETURN;
END_IF

out := ULINT_TO_TOD(in);
TryConvert_ULINT_TO_TOD := TRUE;

END_FUNCTION

// ---- mobject-converters/Converters/ULINT_TO_/TryConvert_ULINT_TO_DATE.TcPOU
FUNCTION TryConvert_ULINT_TO_DATE : BOOL
VAR_INPUT
	in : ULINT;
	out : REFERENCE TO DATE;
END_VAR

IF in > DatatypeLimits.MAX_VALUE_OF_ULINT_WHICH_CAN_BE_HELD_IN_A_DATE THEN
	RETURN;
END_IF

out := ULINT_TO_DATE(in);
TryConvert_ULINT_TO_DATE := TRUE;

END_FUNCTION

// ---- mobject-converters/Converters/UINT_TO_/TryConvert_UINT_TO_BOOL.TcPOU
FUNCTION TryConvert_UINT_TO_BOOL : BOOL
VAR_INPUT
	in : UINT;
	out : REFERENCE TO BOOL;
END_VAR

out := UINT_TO_BOOL(in);
TryConvert_UINT_TO_BOOL := TRUE;

END_FUNCTION

// ---- mobject-converters/Converters/UINT_TO_/TryConvert_UINT_TO_DWORD.TcPOU
FUNCTION TryConvert_UINT_TO_DWORD : BOOL
VAR_INPUT
	in : UINT;
	out : REFERENCE TO DWORD;
END_VAR

out := UINT_TO_DWORD(in);
TryConvert_UINT_TO_DWORD := TRUE;

END_FUNCTION

// ---- mobject-converters/Converters/UINT_TO_/TryConvert_UINT_TO_SINT.TcPOU
FUNCTION TryConvert_UINT_TO_SINT : BOOL
VAR_INPUT
	in : UINT;
	out : REFERENCE TO SINT;
END_VAR

IF in > DatatypeLimits.MAX_VALUE_OF_UINT_WHICH_CAN_BE_HELD_IN_A_SINT THEN
	RETURN;
END_IF

out := UINT_TO_SINT(in);
TryConvert_UINT_TO_SINT := TRUE;

END_FUNCTION

// ---- mobject-converters/Converters/UINT_TO_/TryConvert_UINT_TO_INT.TcPOU
FUNCTION TryConvert_UINT_TO_INT : BOOL
VAR_INPUT
	in : UINT;
	out : REFERENCE TO INT;
END_VAR

IF in > DatatypeLimits.MAX_VALUE_OF_UINT_WHICH_CAN_BE_HELD_IN_A_INT THEN
	RETURN;
END_IF

out := UINT_TO_INT(in);
TryConvert_UINT_TO_INT := TRUE;

END_FUNCTION

// ---- mobject-converters/Converters/UINT_TO_/TryConvert_UINT_TO_LINT.TcPOU
FUNCTION TryConvert_UINT_TO_LINT : BOOL
VAR_INPUT
	in : UINT;
	out : REFERENCE TO LINT;
END_VAR

out := UINT_TO_LINT(in);
TryConvert_UINT_TO_LINT := TRUE;

END_FUNCTION

// ---- mobject-converters/Converters/UINT_TO_/TryConvert_UINT_TO_UINT.TcPOU
FUNCTION TryConvert_UINT_TO_UINT : BOOL
VAR_INPUT
	in : UINT;
	out : REFERENCE TO UINT;
END_VAR

out := in;
TryConvert_UINT_TO_UINT := TRUE;

END_FUNCTION

// ---- mobject-converters/Converters/UINT_TO_/TryConvert_UINT_TO_UDINT.TcPOU
FUNCTION TryConvert_UINT_TO_UDINT : BOOL
VAR_INPUT
	in : UINT;
	out : REFERENCE TO UDINT;
END_VAR

out := UINT_TO_UDINT(in);
TryConvert_UINT_TO_UDINT := TRUE;

END_FUNCTION

// ---- mobject-converters/Converters/UINT_TO_/TryConvert_UINT_TO_REAL.TcPOU
FUNCTION TryConvert_UINT_TO_REAL : BOOL
VAR_INPUT
	in : UINT;
	out : REFERENCE TO REAL;
END_VAR

out := UINT_TO_REAL(in);
TryConvert_UINT_TO_REAL := TRUE;

END_FUNCTION

// ---- mobject-converters/Converters/UINT_TO_/TryConvert_UINT_TO_LREAL.TcPOU
FUNCTION TryConvert_UINT_TO_LREAL : BOOL
VAR_INPUT
	in : UINT;
	out : REFERENCE TO LREAL;
END_VAR

out := UINT_TO_LREAL(in);
TryConvert_UINT_TO_LREAL := TRUE;

END_FUNCTION

// ---- mobject-converters/Converters/UINT_TO_/TryConvert_UINT_TO_TIME.TcPOU
FUNCTION TryConvert_UINT_TO_TIME : BOOL
VAR_INPUT
	in : UINT;
	out : REFERENCE TO TIME;
END_VAR

out := UINT_TO_TIME(in);
TryConvert_UINT_TO_TIME := TRUE;

END_FUNCTION

// ---- mobject-converters/Converters/UINT_TO_/TryConvert_UINT_TO_TOD.TcPOU
FUNCTION TryConvert_UINT_TO_TOD : BOOL
VAR_INPUT
	in : UINT;
	out : REFERENCE TO TOD;
END_VAR

out := UINT_TO_TOD(in);
TryConvert_UINT_TO_TOD := TRUE;

END_FUNCTION

// ---- mobject-converters/Converters/UINT_TO_/TryConvert_UINT_TO_DATE.TcPOU
FUNCTION TryConvert_UINT_TO_DATE : BOOL
VAR_INPUT
	in : UINT;
	out : REFERENCE TO DATE;
END_VAR

out := UINT_TO_DATE(in);
TryConvert_UINT_TO_DATE := TRUE;

END_FUNCTION

// ---- mobject-converters/Converters/USINT_TO_/TryConvert_USINT_TO_WORD.TcPOU
FUNCTION TryConvert_USINT_TO_WORD : BOOL
VAR_INPUT
	in : USINT;
	out : REFERENCE TO WORD;
END_VAR

out := USINT_TO_WORD(in);
TryConvert_USINT_TO_WORD := TRUE;

END_FUNCTION

// ---- mobject-converters/Converters/USINT_TO_/TryConvert_USINT_TO_DWORD.TcPOU
FUNCTION TryConvert_USINT_TO_DWORD : BOOL
VAR_INPUT
	in : USINT;
	out : REFERENCE TO DWORD;
END_VAR

out := USINT_TO_DWORD(in);
TryConvert_USINT_TO_DWORD := TRUE;

END_FUNCTION

// ---- mobject-converters/Converters/USINT_TO_/TryConvert_USINT_TO_SINT.TcPOU
FUNCTION TryConvert_USINT_TO_SINT : BOOL
VAR_INPUT
	in : USINT;
	out : REFERENCE TO SINT;
END_VAR

IF in > DatatypeLimits.MAX_VALUE_OF_USINT_WHICH_CAN_BE_HELD_IN_A_SINT THEN
	RETURN;
END_IF

out := USINT_TO_SINT(in);
TryConvert_USINT_TO_SINT := TRUE;

END_FUNCTION

// ---- mobject-converters/Converters/USINT_TO_/TryConvert_USINT_TO_LINT.TcPOU
FUNCTION TryConvert_USINT_TO_LINT : BOOL
VAR_INPUT
	in : USINT;
	out : REFERENCE TO LINT;
END_VAR

out := USINT_TO_LINT(in);
TryConvert_USINT_TO_LINT := TRUE;

END_FUNCTION

// ---- mobject-converters/Converters/USINT_TO_/TryConvert_USINT_TO_USINT.TcPOU
FUNCTION TryConvert_USINT_TO_USINT : BOOL
VAR_INPUT
	in : USINT;
	out : REFERENCE TO USINT;
END_VAR

out := in;
TryConvert_USINT_TO_USINT := TRUE;

END_FUNCTION

// ---- mobject-converters/Converters/USINT_TO_/TryConvert_USINT_TO_UDINT.TcPOU
FUNCTION TryConvert_USINT_TO_UDINT : BOOL
VAR_INPUT
	in : USINT;
	out : REFERENCE TO UDINT;
END_VAR

out := USINT_TO_UDINT(in);
TryConvert_USINT_TO_UDINT := TRUE;

END_FUNCTION

// ---- mobject-converters/Converters/USINT_TO_/TryConvert_USINT_TO_REAL.TcPOU
FUNCTION TryConvert_USINT_TO_REAL : BOOL
VAR_INPUT
	in : USINT;
	out : REFERENCE TO REAL;
END_VAR

out := USINT_TO_REAL(in);
TryConvert_USINT_TO_REAL := TRUE;

END_FUNCTION

// ---- mobject-converters/Converters/USINT_TO_/TryConvert_USINT_TO_LREAL.TcPOU
FUNCTION TryConvert_USINT_TO_LREAL : BOOL
VAR_INPUT
	in : USINT;
	out : REFERENCE TO LREAL;
END_VAR

out := USINT_TO_LREAL(in);
TryConvert_USINT_TO_LREAL := TRUE;

END_FUNCTION

// ---- mobject-converters/Converters/USINT_TO_/TryConvert_USINT_TO_TIME.TcPOU
FUNCTION TryConvert_USINT_TO_TIME : BOOL
VAR_INPUT
	in : USINT;
	out : REFERENCE TO TIME;
END_VAR

out := USINT_TO_TIME(in);
TryConvert_USINT_TO_TIME := TRUE;

END_FUNCTION

// ---- mobject-converters/Converters/USINT_TO_/TryConvert_USINT_TO_DATE.TcPOU
FUNCTION TryConvert_USINT_TO_DATE : BOOL
VAR_INPUT
	in : USINT;
	out : REFERENCE TO DATE;
END_VAR

out := USINT_TO_DATE(in);
TryConvert_USINT_TO_DATE := TRUE;

END_FUNCTION

// ---- mobject-converters/Converters/USINT_TO_/TryConvert_USINT_TO_STRING.TcPOU
FUNCTION TryConvert_USINT_TO_STRING : BOOL
VAR_INPUT
	in : USINT;
	out : REFERENCE TO STRING;
END_VAR

out := USINT_TO_STRING(in);
TryConvert_USINT_TO_STRING := TRUE;

END_FUNCTION

// ---- mobject-converters/Converters/DWORD_TO_/TryConvert_DWORD_TO_BYTE.TcPOU
FUNCTION TryConvert_DWORD_TO_BYTE : BOOL
VAR_INPUT
	in : DWORD;
	out : REFERENCE TO BYTE;
END_VAR

IF in > DatatypeLimits.MAX_VALUE_OF_DWORD_WHICH_CAN_BE_HELD_IN_A_BYTE THEN
	RETURN;
END_IF

out := DWORD_TO_BYTE(in);
TryConvert_DWORD_TO_BYTE := TRUE;

END_FUNCTION

// ---- mobject-converters/Converters/DWORD_TO_/TryConvert_DWORD_TO_DWORD.TcPOU
FUNCTION TryConvert_DWORD_TO_DWORD : BOOL
VAR_INPUT
	in : DWORD;
	out : REFERENCE TO DWORD;
END_VAR

out := in;
TryConvert_DWORD_TO_DWORD := TRUE;

END_FUNCTION

// ---- mobject-converters/Converters/DWORD_TO_/TryConvert_DWORD_TO_LWORD.TcPOU
FUNCTION TryConvert_DWORD_TO_LWORD : BOOL
VAR_INPUT
	in : DWORD;
	out : REFERENCE TO LWORD;
END_VAR

out := DWORD_TO_LWORD(in);
TryConvert_DWORD_TO_LWORD := TRUE;

END_FUNCTION

// ---- mobject-converters/Converters/DWORD_TO_/TryConvert_DWORD_TO_INT.TcPOU
FUNCTION TryConvert_DWORD_TO_INT : BOOL
VAR_INPUT
	in : DWORD;
	out : REFERENCE TO INT;
END_VAR

IF in > DatatypeLimits.MAX_VALUE_OF_DWORD_WHICH_CAN_BE_HELD_IN_A_INT THEN
	RETURN;
END_IF

out := DWORD_TO_INT(in);
TryConvert_DWORD_TO_INT := TRUE;

END_FUNCTION

// ---- mobject-converters/Converters/DWORD_TO_/TryConvert_DWORD_TO_DINT.TcPOU
FUNCTION TryConvert_DWORD_TO_DINT : BOOL
VAR_INPUT
	in : DWORD;
	out : REFERENCE TO DINT;
END_VAR

IF in > DatatypeLimits.MAX_VALUE_OF_DWORD_WHICH_CAN_BE_HELD_IN_A_DINT THEN
	RETURN;
END_IF

out := DWORD_TO_DINT(in);
TryConvert_DWORD_TO_DINT := TRUE;

END_FUNCTION

// ---- mobject-converters/Converters/DWORD_TO_/TryConvert_DWORD_TO_LINT.TcPOU
FUNCTION TryConvert_DWORD_TO_LINT : BOOL
VAR_INPUT
	in : DWORD;
	out : REFERENCE TO LINT;
END_VAR

out := DWORD_TO_LINT(in);
TryConvert_DWORD_TO_LINT := TRUE;

END_FUNCTION

// ---- mobject-converters/Converters/DWORD_TO_/TryConvert_DWORD_TO_USINT.TcPOU
FUNCTION TryConvert_DWORD_TO_USINT : BOOL
VAR_INPUT
	in : DWORD;
	out : REFERENCE TO USINT;
END_VAR

IF in > DatatypeLimits.MAX_VALUE_OF_DWORD_WHICH_CAN_BE_HELD_IN_A_USINT THEN
	RETURN;
END_IF

out := DWORD_TO_USINT(in);
TryConvert_DWORD_TO_USINT := TRUE;

END_FUNCTION

// ---- mobject-converters/Converters/DWORD_TO_/TryConvert_DWORD_TO_REAL.TcPOU
FUNCTION TryConvert_DWORD_TO_REAL : BOOL
VAR_INPUT
	in : DWORD;
	out : REFERENCE TO REAL;
END_VAR

out := DWORD_TO_REAL(in);
TryConvert_DWORD_TO_REAL := TRUE;

END_FUNCTION

// ---- mobject-converters/Converters/DWORD_TO_/TryConvert_DWORD_TO_TIME.TcPOU
FUNCTION TryConvert_DWORD_TO_TIME : BOOL
VAR_INPUT
	in : DWORD;
	out : REFERENCE TO TIME;
END_VAR

out := DWORD_TO_TIME(in);
TryConvert_DWORD_TO_TIME := TRUE;

END_FUNCTION

// ---- mobject-converters/Converters/DWORD_TO_/TryConvert_DWORD_TO_TOD.TcPOU
FUNCTION TryConvert_DWORD_TO_TOD : BOOL
VAR_INPUT
	in : DWORD;
	out : REFERENCE TO TOD;
END_VAR

IF in > DatatypeLimits.MAX_VALUE_OF_DWORD_WHICH_CAN_BE_HELD_IN_A_TOD THEN
	RETURN;
END_IF

out := DWORD_TO_TOD(in);
TryConvert_DWORD_TO_TOD := TRUE;

END_FUNCTION

// ---- mobject-converters/Converters/DWORD_TO_/TryConvert_DWORD_TO_DATE.TcPOU
FUNCTION TryConvert_DWORD_TO_DATE : BOOL
VAR_INPUT
	in : DWORD;
	out : REFERENCE TO DATE;
END_VAR

out := DWORD_TO_DATE(in);
TryConvert_DWORD_TO_DATE := TRUE;

END_FUNCTION

// ---- mobject-converters/Converters/DWORD_TO_/TryConvert_DWORD_TO_DT.TcPOU
FUNCTION TryConvert_DWORD_TO_DT : BOOL
VAR_INPUT
	in : DWORD;
	out : REFERENCE TO DT;
END_VAR

out := DWORD_TO_DT(in);
TryConvert_DWORD_TO_DT := TRUE;

END_FUNCTION

// ---- mobject-converters/Converters/DWORD_TO_/TryConvert_DWORD_TO_STRING.TcPOU
FUNCTION TryConvert_DWORD_TO_STRING : BOOL
VAR_INPUT
	in : DWORD;
	out : REFERENCE TO STRING;
END_VAR

out := DWORD_TO_STRING(in);
TryConvert_DWORD_TO_STRING := TRUE;

END_FUNCTION

// ---- mobject-converters/Converters/WORD_TO_/TryConvert_WORD_TO_BYTE.TcPOU
FUNCTION TryConvert_WORD_TO_BYTE : BOOL
VAR_INPUT
	in : WORD;
	out : REFERENCE TO BYTE;
END_VAR

IF in > DatatypeLimits.MAX_VALUE_OF_WORD_WHICH_CAN_BE_HELD_IN_A_BYTE THEN
	RETURN;
END_IF

out := WORD_TO_BYTE(in);
TryConvert_WORD_TO_BYTE := TRUE;

END_FUNCTION

// ---- mobject-converters/Converters/WORD_TO_/TryConvert_WORD_TO_WORD.TcPOU
FUNCTION TryConvert_WORD_TO_WORD : BOOL
VAR_INPUT
	in : WORD;
	out : REFERENCE TO WORD;
END_VAR

out := in;
TryConvert_WORD_TO_WORD := TRUE;

END_FUNCTION

// ---- mobject-converters/Converters/WORD_TO_/TryConvert_WORD_TO_DWORD.TcPOU
FUNCTION TryConvert_WORD_TO_DWORD : BOOL
VAR_INPUT
	in : WORD;
	out : REFERENCE TO DWORD;
END_VAR

out := WORD_TO_DWORD(in);
TryConvert_WORD_TO_DWORD := TRUE;

END_FUNCTION

// ---- mobject-converters/Converters/WORD_TO_/TryConvert_WORD_TO_INT.TcPOU
FUNCTION TryConvert_WORD_TO_INT : BOOL
VAR_INPUT
	in : WORD;
	out : REFERENCE TO INT;
END_VAR

IF in > DatatypeLimits.MAX_VALUE_OF_WORD_WHICH_CAN_BE_HELD_IN_A_INT THEN
	RETURN;
END_IF

out := WORD_TO_INT(in);
TryConvert_WORD_TO_INT := TRUE;

END_FUNCTION

// ---- mobject-converters/Converters/WORD_TO_/TryConvert_WORD_TO_DINT.TcPOU
FUNCTION TryConvert_WORD_TO_DINT : BOOL
VAR_INPUT
	in : WORD;
	out : REFERENCE TO DINT;
END_VAR

out := WORD_TO_DINT(in);
TryConvert_WORD_TO_DINT := TRUE;

END_FUNCTION

// ---- mobject-converters/Converters/WORD_TO_/TryConvert_WORD_TO_UINT.TcPOU
FUNCTION TryConvert_WORD_TO_UINT : BOOL
VAR_INPUT
	in : WORD;
	out : REFERENCE TO UINT;
END_VAR

out := WORD_TO_UINT(in);
TryConvert_WORD_TO_UINT := TRUE;

END_FUNCTION

// ---- mobject-converters/Converters/WORD_TO_/TryConvert_WORD_TO_UDINT.TcPOU
FUNCTION TryConvert_WORD_TO_UDINT : BOOL
VAR_INPUT
	in : WORD;
	out : REFERENCE TO UDINT;
END_VAR

out := WORD_TO_UDINT(in);
TryConvert_WORD_TO_UDINT := TRUE;

END_FUNCTION

// ---- mobject-converters/Converters/WORD_TO_/TryConvert_WORD_TO_LREAL.TcPOU
FUNCTION TryConvert_WORD_TO_LREAL : BOOL
VAR_INPUT
	in : WORD;
	out : REFERENCE TO LREAL;
END_VAR

out := WORD_TO_LREAL(in);
TryConvert_WORD_TO_LREAL := TRUE;

END_FUNCTION

// ---- mobject-converters/Converters/WORD_TO_/TryConvert_WORD_TO_TOD.TcPOU
FUNCTION TryConvert_WORD_TO_TOD : BOOL
VAR_INPUT
	in : WORD;
	out : REFERENCE TO TOD;
END_VAR

out := WORD_TO_TOD(in);
TryConvert_WORD_TO_TOD := TRUE;

END_FUNCTION

// ---- mobject-converters/Converters/WORD_TO_/TryConvert_WORD_TO_DATE.TcPOU
FUNCTION TryConvert_WORD_TO_DATE : BOOL
VAR_INPUT
	in : WORD;
	out : REFERENCE TO DATE;
END_VAR

out := WORD_TO_DATE(in);
TryConvert_WORD_TO_DATE := TRUE;

END_FUNCTION

// ---- mobject-converters/Converters/WORD_TO_/TryConvert_WORD_TO_STRING.TcPOU
FUNCTION TryConvert_WORD_TO_STRING : BOOL
VAR_INPUT
	in : WORD;
	out : REFERENCE TO STRING;
END_VAR

out := WORD_TO_STRING(in);
TryConvert_WORD_TO_STRING := TRUE;

END_FUNCTION

// ---- mobject-converters/Converters/DATE_TO_/TryConvert_DATE_TO_BOOL.TcPOU
FUNCTION TryConvert_DATE_TO_BOOL : BOOL
VAR_INPUT
	in : DATE;
	out : REFERENCE TO BOOL;
END_VAR

out := DATE_TO_BOOL(in);
TryConvert_DATE_TO_BOOL := TRUE;

END_FUNCTION

// ---- mobject-converters/Converters/DATE_TO_/TryConvert_DATE_TO_BYTE.TcPOU
FUNCTION TryConvert_DATE_TO_BYTE : BOOL
VAR_INPUT
	in : DATE;
	out : REFERENCE TO BYTE;
END_VAR

IF in > DatatypeLimits.MAX_VALUE_OF_DATE_WHICH_CAN_BE_HELD_IN_A_BYTE THEN
	RETURN;
END_IF

out := DATE_TO_BYTE(in);
TryConvert_DATE_TO_BYTE := TRUE;

END_FUNCTION

// ---- mobject-converters/Converters/DATE_TO_/TryConvert_DATE_TO_Destination.TcPOU
FUNCTION TryConvert_DATE_TO_Destination : BOOL
VAR_INPUT
	in : DATE;
	out : ANY;
END_VAR
VAR
	convertResult : BOOL := FALSE;
	convertAddress : PVOID;
	_BOOL : BOOL;
	_BYTE : BYTE;
	_WORD : WORD;
	_DWORD : DWORD;
	_LWORD : LWORD;
	_SINT : SINT;
	_INT : INT;
	_DINT : DINT;
	_LINT : LINT;
	_USINT : USINT;
	_UINT : UINT;
	_UDINT : UDINT;
	_ULINT : ULINT;
	_REAL : REAL;
	_LREAL : LREAL;
	_TIME : TIME;
	_TOD : TOD;
	_DATE : DATE;
	_DT : DT;
	_STRING : STRING;
END_VAR

CASE out.TypeClass OF
	__SYSTEM.TYPE_CLASS.TYPE_BOOL:
	
	convertResult := TryConvert_DATE_TO_BOOL(in, _BOOL);
	IF convertResult THEN
		convertAddress := ADR(_BOOL);
	END_IF
	
	__SYSTEM.TYPE_CLASS.TYPE_BYTE:
	
	convertResult := TryConvert_DATE_TO_BYTE(in, _BYTE);
	IF convertResult THEN
		convertAddress := ADR(_BYTE);
	END_IF
	
	__SYSTEM.TYPE_CLASS.TYPE_WORD:
	
	convertResult := TryConvert_DATE_TO_WORD(in, _WORD);
	IF convertResult THEN
		convertAddress := ADR(_WORD);
	END_IF
	
	__SYSTEM.TYPE_CLASS.TYPE_DWORD:
	
	convertResult := TryConvert_DATE_TO_DWORD(in, _DWORD);
	IF convertResult THEN
		convertAddress := ADR(_DWORD);
	END_IF
	
	__SYSTEM.TYPE_CLASS.TYPE_LWORD:
	
	convertResult := TryConvert_DATE_TO_LWORD(in, _LWORD);
	IF convertResult THEN
		convertAddress := ADR(_LWORD);
	END_IF
	
	__SYSTEM.TYPE_CLASS.TYPE_SINT:
	
	convertResult := TryConvert_DATE_TO_SINT(in, _SINT);
	IF convertResult THEN
		convertAddress := ADR(_SINT);
	END_IF
	
	__SYSTEM.TYPE_CLASS.TYPE_INT:
	
	convertResult := TryConvert_DATE_TO_INT(in, _INT);
	IF convertResult THEN
		convertAddress := ADR(_INT);
	END_IF
	
	__SYSTEM.TYPE_CLASS.TYPE_DINT:
	
	convertResult := TryConvert_DATE_TO_DINT(in, _DINT);
	IF convertResult THEN
		convertAddress := ADR(_DINT);
	END_IF
	
	__SYSTEM.TYPE_CLASS.TYPE_LINT:
	
	convertResult := TryConvert_DATE_TO_LINT(in, _LINT);
	IF convertResult THEN
		convertAddress := ADR(_LINT);
	END_IF
	
	__SYSTEM.TYPE_CLASS.TYPE_USINT:
	
	convertResult := TryConvert_DATE_TO_USINT(in, _USINT);
	IF convertResult THEN
		convertAddress := ADR(_USINT);
	END_IF
	
	__SYSTEM.TYPE_CLASS.TYPE_UINT:
	
	convertResult := TryConvert_DATE_TO_UINT(in, _UINT);
	IF convertResult THEN
		convertAddress := ADR(_UINT);
	END_IF
	
	__SYSTEM.TYPE_CLASS.TYPE_UDINT:
	
	convertResult := TryConvert_DATE_TO_UDINT(in, _UDINT);
	IF convertResult THEN
		convertAddress := ADR(_UDINT);
	END_IF
	
	__SYSTEM.TYPE_CLASS.TYPE_ULINT:
	
	convertResult := TryConvert_DATE_TO_ULINT(in, _ULINT);
	IF convertResult THEN
		convertAddress := ADR(_ULINT);
	END_IF
	
	__SYSTEM.TYPE_CLASS.TYPE_REAL:
	
	convertResult := TryConvert_DATE_TO_REAL(in, _REAL);
	IF convertResult THEN
		convertAddress := ADR(_REAL);
	END_IF
	
	__SYSTEM.TYPE_CLASS.TYPE_LREAL:
	
	convertResult := TryConvert_DATE_TO_LREAL(in, _LREAL);
	IF convertResult THEN
		convertAddress := ADR(_LREAL);
	END_IF
	
	__SYSTEM.TYPE_CLASS.TYPE_TIME:
	
	convertResult := TryConvert_DATE_TO_TIME(in, _TIME);
	IF convertResult THEN
		convertAddress := ADR(_TIME);
	END_IF
	
	__SYSTEM.TYPE_CLASS.TYPE_TIMEOFDAY:
	
	convertResult := TryConvert_DATE_TO_TOD(in, _TOD);
	IF convertResult THEN
		convertAddress := ADR(_TOD);
	END_IF
	
	__SYSTEM.TYPE_CLASS.TYPE_DATE:
	
	convertResult := TryConvert_DATE_TO_DATE(in, _DATE);
	IF convertResult THEN
		convertAddress := ADR(_DATE);
	END_IF
	
	__SYSTEM.TYPE_CLASS.TYPE_DATEANDTIME:
	
	convertResult := TryConvert_DATE_TO_DT(in, _DT);
	IF convertResult THEN
		convertAddress := ADR(_DT);
	END_IF
	
	__SYSTEM.TYPE_CLASS.TYPE_STRING:
	
	convertResult := TryConvert_DATE_TO_STRING(in, _STRING);
	IF convertResult THEN
		convertAddress := ADR(_STRING);
	END_IF
	
END_CASE

IF convertResult THEN
	memcpy(out.pValue,convertAddress,DINT_TO_UDINT(out.diSize));
END_IF

TryConvert_DATE_TO_Destination := convertResult;

END_FUNCTION

// ---- mobject-converters/Converters/DATE_TO_/TryConvert_DATE_TO_SINT.TcPOU
FUNCTION TryConvert_DATE_TO_SINT : BOOL
VAR_INPUT
	in : DATE;
	out : REFERENCE TO SINT;
END_VAR

IF in > DatatypeLimits.MAX_VALUE_OF_DATE_WHICH_CAN_BE_HELD_IN_A_SINT THEN
	RETURN;
END_IF

out := DATE_TO_SINT(in);
TryConvert_DATE_TO_SINT := TRUE;

END_FUNCTION

// ---- mobject-converters/Converters/DATE_TO_/TryConvert_DATE_TO_INT.TcPOU
FUNCTION TryConvert_DATE_TO_INT : BOOL
VAR_INPUT
	in : DATE;
	out : REFERENCE TO INT;
END_VAR

IF in > DatatypeLimits.MAX_VALUE_OF_DATE_WHICH_CAN_BE_HELD_IN_A_INT THEN
	RETURN;
END_IF

out := DATE_TO_INT(in);
TryConvert_DATE_TO_INT := TRUE;

END_FUNCTION

// ---- mobject-converters/Converters/DATE_TO_/TryConvert_DATE_TO_DINT.TcPOU
FUNCTION TryConvert_DATE_TO_DINT : BOOL
VAR_INPUT
	in : DATE;
	out : REFERENCE TO DINT;
END_VAR

IF in > DatatypeLimits.MAX_VALUE_OF_DATE_WHICH_CAN_BE_HELD_IN_A_DINT THEN
	RETURN;
END_IF

out := DATE_TO_DINT(in);
TryConvert_DATE_TO_DINT := TRUE;

END_FUNCTION

// ---- mobject-converters/Converters/DATE_TO_/TryConvert_DATE_TO_LINT.TcPOU
FUNCTION TryConvert_DATE_TO_LINT : BOOL
VAR_INPUT
	in : DATE;
	out : REFERENCE TO LINT;
END_VAR

out := DATE_TO_LINT(in);
TryConvert_DATE_TO_LINT := TRUE;

END_FUNCTION

// ---- mobject-converters/Converters/DATE_TO_/TryConvert_DATE_TO_UDINT.TcPOU
FUNCTION TryConvert_DATE_TO_UDINT : BOOL
VAR_INPUT
	in : DATE;
	out : REFERENCE TO UDINT;
END_VAR

out := DATE_TO_UDINT(in);
TryConvert_DATE_TO_UDINT := TRUE;

END_FUNCTION

// ---- mobject-converters/Converters/DATE_TO_/TryConvert_DATE_TO_TIME.TcPOU
FUNCTION TryConvert_DATE_TO_TIME : BOOL
VAR_INPUT
	in : DATE;
	out : REFERENCE TO TIME;
END_VAR

IF in > DatatypeLimits.MAX_VALUE_OF_DATE_WHICH_CAN_BE_HELD_IN_A_TIME THEN
	RETURN;
END_IF

out := DATE_TO_TIME(in);
TryConvert_DATE_TO_TIME := TRUE;

END_FUNCTION

// ---- mobject-converters/Converters/DINT_TO_/TryConvert_DINT_TO_TIME.TcPOU
FUNCTION TryConvert_DINT_TO_TIME : BOOL
VAR_INPUT
	in : DINT;
	out : REFERENCE TO TIME;
END_VAR

IF in < DatatypeLimits.MIN_VALUE_OF_DINT_WHICH_CAN_BE_HELD_IN_A_TIME THEN
	RETURN;
END_IF

out := DINT_TO_TIME(in);
TryConvert_DINT_TO_TIME := TRUE;

END_FUNCTION

// ---- mobject-converters/Converters/INT_TO_/TryConvert_INT_TO_DATE.TcPOU
FUNCTION TryConvert_INT_TO_DATE : BOOL
VAR_INPUT
	in : INT;
	out : REFERENCE TO DATE;
END_VAR

IF in < DatatypeLimits.MIN_VALUE_OF_INT_WHICH_CAN_BE_HELD_IN_A_DATE THEN
	RETURN;
END_IF

out := INT_TO_DATE(in);
TryConvert_INT_TO_DATE := TRUE;

END_FUNCTION

// ---- mobject-converters/Converters/INT_TO_/TryConvert_INT_TO_TIME.TcPOU
FUNCTION TryConvert_INT_TO_TIME : BOOL
VAR_INPUT
	in : INT;
	out : REFERENCE TO TIME;
END_VAR

IF in < DatatypeLimits.MIN_VALUE_OF_INT_WHICH_CAN_BE_HELD_IN_A_TIME THEN
	RETURN;
END_IF

out := INT_TO_TIME(in);
TryConvert_INT_TO_TIME := TRUE;

END_FUNCTION

// ---- mobject-converters/Converters/LINT_TO_/TryConvert_LINT_TO_DATE.TcPOU
FUNCTION TryConvert_LINT_TO_DATE : BOOL
VAR_INPUT
	in : LINT;
	out : REFERENCE TO DATE;
END_VAR

IF in > DatatypeLimits.MAX_VALUE_OF_LINT_WHICH_CAN_BE_HELD_IN_A_DATE THEN
	RETURN;
END_IF

IF in < DatatypeLimits.MIN_VALUE_OF_LINT_WHICH_CAN_BE_HELD_IN_A_DATE THEN
	RETURN;
END_IF

out := LINT_TO_DATE(in);
TryConvert_LINT_TO_DATE := TRUE;

END_FUNCTION

// ---- mobject-converters/Converters/LINT_TO_/TryConvert_LINT_TO_TIME.TcPOU
FUNCTION TryConvert_LINT_TO_TIME : BOOL
VAR_INPUT
	in : LINT;
	out : REFERENCE TO TIME;
END_VAR

IF in > DatatypeLimits.MAX_VALUE_OF_LINT_WHICH_CAN_BE_HELD_IN_A_TIME THEN
	RETURN;
END_IF

IF in < DatatypeLimits.MIN_VALUE_OF_LINT_WHICH_CAN_BE_HELD_IN_A_TIME THEN
	RETURN;
END_IF

out := LINT_TO_TIME(in);
TryConvert_LINT_TO_TIME := TRUE;

END_FUNCTION

// ---- mobject-converters/Converters/LREAL_TO_/TryConvert_LREAL_TO_DATE.TcPOU
FUNCTION TryConvert_LREAL_TO_DATE : BOOL
VAR_INPUT
	in : LREAL;
	out : REFERENCE TO DATE;
END_VAR

IF in > DatatypeLimits.MAX_VALUE_OF_LREAL_WHICH_CAN_BE_HELD_IN_A_DATE THEN
	RETURN;
END_IF

IF in < DatatypeLimits.MIN_VALUE_OF_LREAL_WHICH_CAN_BE_HELD_IN_A_DATE THEN
	RETURN;
END_IF

out := LREAL_TO_DATE(in);
TryConvert_LREAL_TO_DATE := TRUE;

END_FUNCTION

// ---- mobject-converters/Converters/LWORD_TO_/TryConvert_LWORD_TO_DATE.TcPOU
FUNCTION TryConvert_LWORD_TO_DATE : BOOL
VAR_INPUT
	in : LWORD;
	out : REFERENCE TO DATE;
END_VAR

IF in > DatatypeLimits.MAX_VALUE_OF_LWORD_WHICH_CAN_BE_HELD_IN_A_DATE THEN
	RETURN;
END_IF

out := LWORD_TO_DATE(in);
TryConvert_LWORD_TO_DATE := TRUE;

END_FUNCTION

// ---- mobject-converters/Converters/REAL_TO_/TryConvert_REAL_TO_DATE.TcPOU
FUNCTION TryConvert_REAL_TO_DATE : BOOL
VAR_INPUT
	in : REAL;
	out : REFERENCE TO DATE;
END_VAR

IF in > DatatypeLimits.MAX_VALUE_OF_REAL_WHICH_CAN_BE_HELD_IN_A_DATE THEN
	RETURN;
END_IF

IF in < DatatypeLimits.MIN_VALUE_OF_REAL_WHICH_CAN_BE_HELD_IN_A_DATE THEN
	RETURN;
END_IF

out := REAL_TO_DATE(in);
TryConvert_REAL_TO_DATE := TRUE;

END_FUNCTION

// ---- mobject-converters/Converters/REAL_TO_/TryConvert_REAL_TO_TIME.TcPOU
FUNCTION TryConvert_REAL_TO_TIME : BOOL
VAR_INPUT
	in : REAL;
	out : REFERENCE TO TIME;
END_VAR

IF in > DatatypeLimits.MAX_VALUE_OF_REAL_WHICH_CAN_BE_HELD_IN_A_TIME THEN
	RETURN;
END_IF

IF in < DatatypeLimits.MIN_VALUE_OF_REAL_WHICH_CAN_BE_HELD_IN_A_TIME THEN
	RETURN;
END_IF

out := REAL_TO_TIME(in);
TryConvert_REAL_TO_TIME := TRUE;

END_FUNCTION

// ---- mobject-converters/Converters/TIME_TO_/TryConvert_TIME_TO_BOOL.TcPOU
FUNCTION TryConvert_TIME_TO_BOOL : BOOL
VAR_INPUT
	in : TIME;
	out : REFERENCE TO BOOL;
END_VAR

out := TIME_TO_BOOL(in);
TryConvert_TIME_TO_BOOL := TRUE;

END_FUNCTION

// ---- mobject-converters/Converters/TIME_TO_/TryConvert_TIME_TO_BYTE.TcPOU
FUNCTION TryConvert_TIME_TO_BYTE : BOOL
VAR_INPUT
	in : TIME;
	out : REFERENCE TO BYTE;
END_VAR

IF in > DatatypeLimits.MAX_VALUE_OF_TIME_WHICH_CAN_BE_HELD_IN_A_BYTE THEN
	RETURN;
END_IF

out := TIME_TO_BYTE(in);
TryConvert_TIME_TO_BYTE := TRUE;

END_FUNCTION

// ---- mobject-converters/Converters/TIME_TO_/TryConvert_TIME_TO_DINT.TcPOU
FUNCTION TryConvert_TIME_TO_DINT : BOOL
VAR_INPUT
	in : TIME;
	out : REFERENCE TO DINT;
END_VAR

IF in > DatatypeLimits.MAX_VALUE_OF_TIME_WHICH_CAN_BE_HELD_IN_A_DINT THEN
	RETURN;
END_IF

out := TIME_TO_DINT(in);
TryConvert_TIME_TO_DINT := TRUE;

END_FUNCTION

// ---- mobject-converters/Converters/TIME_TO_/TryConvert_TIME_TO_DWORD.TcPOU
FUNCTION TryConvert_TIME_TO_DWORD : BOOL
VAR_INPUT
	in : TIME;
	out : REFERENCE TO DWORD;
END_VAR

out := TIME_TO_DWORD(in);
TryConvert_TIME_TO_DWORD := TRUE;

END_FUNCTION

// ---- mobject-converters/Converters/TIME_TO_/TryConvert_TIME_TO_INT.TcPOU
FUNCTION TryConvert_TIME_TO_INT : BOOL
VAR_INPUT
	in : TIME;
	out : REFERENCE TO INT;
END_VAR

IF in > DatatypeLimits.MAX_VALUE_OF_TIME_WHICH_CAN_BE_HELD_IN_A_INT THEN
	RETURN;
END_IF

out := TIME_TO_INT(in);
TryConvert_TIME_TO_INT := TRUE;

END_FUNCTION

// ---- mobject-converters/Converters/TIME_TO_/TryConvert_TIME_TO_LWORD.TcPOU
FUNCTION TryConvert_TIME_TO_LWORD : BOOL
VAR_INPUT
	in : TIME;
	out : REFERENCE TO LWORD;
END_VAR

out := TIME_TO_LWORD(in);
TryConvert_TIME_TO_LWORD := TRUE;

END_FUNCTION

// ---- mobject-converters/Converters/TIME_TO_/TryConvert_TIME_TO_REAL.TcPOU
FUNCTION TryConvert_TIME_TO_REAL : BOOL
VAR_INPUT
	in : TIME;
	out : REFERENCE TO REAL;
END_VAR

out := TIME_TO_REAL(in);
TryConvert_TIME_TO_REAL := TRUE;

END_FUNCTION

// ---- mobject-converters/Converters/TIME_TO_/TryConvert_TIME_TO_SINT.TcPOU
FUNCTION TryConvert_TIME_TO_SINT : BOOL
VAR_INPUT
	in : TIME;
	out : REFERENCE TO SINT;
END_VAR

IF in > DatatypeLimits.MAX_VALUE_OF_TIME_WHICH_CAN_BE_HELD_IN_A_SINT THEN
	RETURN;
END_IF

out := TIME_TO_SINT(in);
TryConvert_TIME_TO_SINT := TRUE;

END_FUNCTION

// ---- mobject-converters/Converters/TIME_TO_/TryConvert_TIME_TO_STRING.TcPOU
FUNCTION TryConvert_TIME_TO_STRING : BOOL
VAR_INPUT
	in : TIME;
	out : REFERENCE TO STRING;
END_VAR

out := TIME_TO_STRING(in);
TryConvert_TIME_TO_STRING := TRUE;

END_FUNCTION

// ---- mobject-converters/Converters/TIME_TO_/TryConvert_TIME_TO_TIME.TcPOU
FUNCTION TryConvert_TIME_TO_TIME : BOOL
VAR_INPUT
	in : TIME;
	out : REFERENCE TO TIME;
END_VAR

out := in;
TryConvert_TIME_TO_TIME := TRUE;

END_FUNCTION

// ---- mobject-converters/Converters/TIME_TO_/TryConvert_TIME_TO_UDINT.TcPOU
FUNCTION TryConvert_TIME_TO_UDINT : BOOL
VAR_INPUT
	in : TIME;
	out : REFERENCE TO UDINT;
END_VAR

out := TIME_TO_UDINT(in);
TryConvert_TIME_TO_UDINT := TRUE;

END_FUNCTION

// ---- mobject-converters/Converters/TIME_TO_/TryConvert_TIME_TO_USINT.TcPOU
FUNCTION TryConvert_TIME_TO_USINT : BOOL
VAR_INPUT
	in : TIME;
	out : REFERENCE TO USINT;
END_VAR

IF in > DatatypeLimits.MAX_VALUE_OF_TIME_WHICH_CAN_BE_HELD_IN_A_USINT THEN
	RETURN;
END_IF

out := TIME_TO_USINT(in);
TryConvert_TIME_TO_USINT := TRUE;

END_FUNCTION

// ---- mobject-converters/Converters/TIME_TO_/TryConvert_TIME_TO_WORD.TcPOU
FUNCTION TryConvert_TIME_TO_WORD : BOOL
VAR_INPUT
	in : TIME;
	out : REFERENCE TO WORD;
END_VAR

IF in > DatatypeLimits.MAX_VALUE_OF_TIME_WHICH_CAN_BE_HELD_IN_A_WORD THEN
	RETURN;
END_IF

out := TIME_TO_WORD(in);
TryConvert_TIME_TO_WORD := TRUE;

END_FUNCTION

// ---- mobject-converters/Converters/UDINT_TO_/TryConvert_UDINT_TO_DATE.TcPOU
FUNCTION TryConvert_UDINT_TO_DATE : BOOL
VAR_INPUT
	in : UDINT;
	out : REFERENCE TO DATE;
END_VAR

out := UDINT_TO_DATE(in);
TryConvert_UDINT_TO_DATE := TRUE;

END_FUNCTION

// ---- mobject-datatypes/DatatypeOperations/Collection/DatatypeOperations.TcPOU
{attribute 'linkalways'} 
{attribute 'no_explicit_call' := 'This FB is a CLASS and must be accessed using methods or properties'}
{attribute 'enable_dynamic_creation'}
FUNCTION_BLOCK DatatypeOperations
VAR
	operations : Stack;
END_VAR

METHOD PUBLIC AddMemoryCopyOperation
VAR_INPUT
	Source : I_Datatype;
	Destination : I_Datatype;
END_VAR
VAR
	operation : I_DatatypeOperation;
END_VAR
operation := CreateMemoryCopyOperation(Source,Destination);
operations.Push(operation);
END_METHOD

METHOD PUBLIC AddSafeMemoryCopyOperation
VAR_INPUT
	Source : I_Datatype;
	Destination : I_Datatype;
END_VAR
VAR
	operation : I_DatatypeOperation;
END_VAR
operation := CreateSafeMemoryCopyOperation(Source,Destination);
operations.Push(operation);
END_METHOD

METHOD PUBLIC AddWriteBitToBoolOperation
VAR_INPUT
	Source : I_BIT;
	Destination : Reference to _BOOL;
END_VAR
VAR
	operation : I_DatatypeOperation;
END_VAR
operation := CreateWriteBitToBoolOperation(Source,Destination);
operations.Push(operation);
END_METHOD

METHOD PUBLIC AddWriteBoolToBitOperation
VAR_INPUT
	Source : REFERENCE TO _BOOL;
	Destination : I_BIT;
END_VAR
VAR
	operation : I_DatatypeOperation;
END_VAR
operation := CreateWriteBoolToBitOperation(Source,Destination);
operations.Push(operation);
END_METHOD

METHOD PUBLIC Clear
VAR
	operation : I_DatatypeOperation;
END_VAR
WHILE operations.TryPop(operation) DO
	operation.Dispose();
END_WHILE
END_METHOD

METHOD PRIVATE CreateMemoryCopyOperation : I_DatatypeOperation
VAR_INPUT
	OperationSource : I_Datatype;
	OperationDestination : I_Datatype;
END_VAR
VAR
	pOperation : POINTER TO MemCopyOperation;
END_VAR
pOperation := __NEW(MemCopyOperation(Source := OperationSource, Destination := OperationDestination));
CreateMemoryCopyOperation := pOperation^;
END_METHOD

METHOD PRIVATE CreateSafeMemoryCopyOperation : I_DatatypeOperation
VAR_INPUT
	OperationSource : I_Datatype;
	OperationDestination : I_Datatype;
END_VAR
VAR
	pOperation : POINTER TO SafeMemCopyOperation;
END_VAR
pOperation := __NEW(SafeMemCopyOperation(Source := OperationSource, Destination := OperationDestination));
CreateSafeMemoryCopyOperation := pOperation^;
END_METHOD

METHOD PRIVATE CreateWriteBitToBoolOperation : I_DatatypeOperation
VAR_INPUT
	OperationSource : I_BIT;
	OperationDestination : REFERENCE TO _BOOL;
END_VAR
VAR
	pOperation : POINTER TO WriteBitToBoolOperation;
END_VAR
pOperation := __NEW(WriteBitToBoolOperation(Source := OperationSource, Destination := OperationDestination));
CreateWriteBitToBoolOperation := pOperation^;
END_METHOD

METHOD PRIVATE CreateWriteBoolToBitOperation : I_DatatypeOperation
VAR_INPUT
	OperationSource : REFERENCE TO _BOOL;
	OperationDestination : I_BIT;
END_VAR
VAR
	pOperation : POINTER TO WriteBoolToBitOperation;
END_VAR
pOperation := __NEW(WriteBoolToBitOperation(Source := OperationSource, Destination := OperationDestination));
CreateWriteBoolToBitOperation := pOperation^;
END_METHOD

METHOD PUBLIC Execute
VAR
	enumerator : I_ForwardEnumerator;
	operation : I_DatatypeOperation;
END_VAR
enumerator := operations.GetEnumerator();

WHILE enumerator.MoveNext() DO
	IF enumerator.TryGet(operation) THEN
		operation.Execute();
	END_IF
END_WHILE

enumerator.Dispose();
END_METHOD

METHOD FB_exit : BOOL
VAR_INPUT
	bInCopyCode : BOOL; // if TRUE, the exit method is called for exiting an instance that is copied afterwards (online change).
END_VAR
IF bInCopyCode THEN
	RETURN;
END_IF

operations.Clear();
END_METHOD

END_FUNCTION_BLOCK

// ---- mobject-datatypes/DatatypeOperations/WriteBitToBoolOperation.TcPOU
{attribute 'linkalways'} 
{attribute 'no_explicit_call' := 'This FB is a CLASS and must be accessed using methods or properties'}
{attribute 'enable_dynamic_creation'}
FUNCTION_BLOCK WriteBitToBoolOperation EXTENDS Disposable IMPLEMENTS I_DatatypeOperation
VAR
	source : I_BIT;
	destination : REFERENCE TO _BOOL;
END_VAR

METHOD Execute
VAR
END_VAR
destination.Value := source.Value;
END_METHOD

METHOD FB_init : BOOL
VAR_INPUT
	bInitRetains : BOOL; // if TRUE, the retain variables are initialized (warm start / cold start)
	bInCopyCode : BOOL;  // if TRUE, the instance afterwards gets moved into the copy code (online change)
	Source : I_BIT;
	Destination : REFERENCE TO _BOOL;
END_VAR
THIS^.source := Source;
THIS^.destination REF= Destination;
END_METHOD

END_FUNCTION_BLOCK

// ---- mobject-datatypes/DatatypeOperations/WriteBoolToBitOperation.TcPOU
{attribute 'linkalways'} 
{attribute 'no_explicit_call' := 'This FB is a CLASS and must be accessed using methods or properties'}
{attribute 'enable_dynamic_creation'}
FUNCTION_BLOCK WriteBoolToBitOperation EXTENDS Disposable IMPLEMENTS I_DatatypeOperation
VAR
	source : REFERENCE TO _BOOL;
	destination : I_BIT;
END_VAR

METHOD Execute
VAR
END_VAR
destination.Value := source.Value;
END_METHOD

METHOD FB_init : BOOL
VAR_INPUT
	bInitRetains : BOOL; // if TRUE, the retain variables are initialized (warm start / cold start)
	bInCopyCode : BOOL;  // if TRUE, the instance afterwards gets moved into the copy code (online change)
	Source : REFERENCE TO _BOOL;
	Destination : I_BIT;
END_VAR
THIS^.source REF= Source;
THIS^.destination := Destination;
END_METHOD

END_FUNCTION_BLOCK

// ---- mobject-datatypes/Primitive/_REFERENCE_TO.TcPOU
{attribute 'linkalways'} 
{attribute 'no_explicit_call' := 'This FB is a CLASS and must be accessed using methods or properties'}
{attribute 'enable_dynamic_creation'}
FUNCTION_BLOCK _REFERENCE_TO EXTENDS Disposable IMPLEMENTS I_REFERENCE_TO
VAR
	nullTarget : _NULL;
	_target : I_Datatype := nullTarget;
END_VAR

METHOD PUBLIC Accept
VAR_INPUT
	Visitor : I_DatatypeVisitor;
END_VAR
Visitor.VisitDatatype(THIS^);
END_METHOD

PROPERTY PUBLIC Address : PVOID
GET
Address := _target.Address;
END_GET
END_PROPERTY

METHOD PUBLIC ClearReference
VAR_INPUT
END_VAR
_target := nullTarget;
END_METHOD

METHOD PUBLIC Clone : I_Datatype
VAR
    pClone : POINTER TO _REFERENCE_TO;
END_VAR
pClone := __NEW(_REFERENCE_TO(RefTo := _target));
Clone := pClone^;
END_METHOD

//FB_Init is always available implicitly and it is used primarily for initialization.
//The return value is not evaluated. For a specific influence, you can also declare the
//methods explicitly and provide additional code there with the standard initialization
//code. You can evaluate the return value.
METHOD FB_Init: BOOL
VAR_INPUT
    bInitRetains: BOOL; // TRUE: the retain variables are initialized (reset warm / reset cold)
    bInCopyCode: BOOL;  // TRUE: the instance will be copied to the copy code afterward (online change)  
	RefTo : I_Datatype; 
END_VAR
IF RefTo = 0 THEN
	RETURN;
END_IF

this^._target := RefTo;
END_METHOD

METHOD PUBLIC IsEquivalentTo : BOOL
VAR_INPUT
	Datatype : I_Datatype;
END_VAR
IsEquivalentTo := _target.IsEquivalentTo(Datatype);
END_METHOD

PROPERTY PUBLIC IsNull : BOOL
GET
IsNull := _target.IsNull;
END_GET
END_PROPERTY

PROPERTY PUBLIC IsUserDefined : BOOL
GET
IsUserDefined := _target.IsUserDefined;
END_GET
END_PROPERTY

PROPERTY PUBLIC IsValidReference : BOOL
GET
IF _target.IsNull THEN
	RETURN;
END_IF

IsValidReference := TRUE;
END_GET
END_PROPERTY

PROPERTY PUBLIC Root : I_Datatype
GET
IF _target.IsNull THEN
	Root := THIS^;
	RETURN;
END_IF

Root := _target.Root;
END_GET
END_PROPERTY

METHOD PUBLIC SerializeTypeWith
VAR_INPUT
	Serializer : I_Serializer;
END_VAR
Serializer.StartObject();
Serializer.AddKeyString('typeName',TypeName);
Serializer.EndObject();
END_METHOD

METHOD PUBLIC SerializeWith
VAR_INPUT
	Serializer : I_Serializer;
END_VAR
_target.SerializeWith(Serializer);
END_METHOD

PROPERTY PUBLIC Size : UDINT
GET
Size := _target.Size;
END_GET
END_PROPERTY

METHOD PUBLIC TryConvertTo : BOOL
VAR_INPUT
	Destination : ANY;
END_VAR
TryConvertTo := _target.TryConvertTo(Destination);
END_METHOD

METHOD PUBLIC TryConvertTo_ : BOOL
VAR_INPUT
	Destination : I_Datatype;
END_VAR
TryConvertTo_ := _target.TryConvertTo_(Destination);
END_METHOD

METHOD PUBLIC TryCopyFrom : BOOL
VAR_INPUT
	Source : I_Datatype;
END_VAR
TryCopyFrom := _target.TryCopyFrom(Source);
END_METHOD

METHOD TryDeserializeFrom : BOOL
VAR_INPUT
	Deserializer : I_Deserializer;
	Feedback : I_DeserializerFeedback;
END_VAR
TryDeserializeFrom := _target.TryDeserializeFrom(Deserializer, Feedback);
END_METHOD

METHOD TryMakeReferenceTo : BOOL
VAR_INPUT
	Target : I_Datatype;
END_VAR
IF Target = 0 THEN
	RETURN;
END_IF

_target := Target;
TryMakeReferenceTo := TRUE;
END_METHOD

METHOD PUBLIC TryResolveAs_ANY : BOOL
VAR_INPUT
	Destination : REFERENCE TO I_ANY;
END_VAR
TryResolveAs_ANY := _target.TryResolveAs_ANY(Destination);
END_METHOD

METHOD PUBLIC TryResolveAs_BIT : BOOL
VAR_INPUT
	Destination : REFERENCE TO I_BIT;
END_VAR
TryResolveAs_BIT := _target.TryResolveAs_BIT(Destination);
END_METHOD

METHOD PUBLIC TryResolveAs_BOOL : BOOL
VAR_INPUT
	Destination : REFERENCE TO I_BOOL;
END_VAR
TryResolveAs_BOOL := _target.TryResolveAs_BOOL(Destination);
END_METHOD

METHOD PUBLIC TryResolveAs_BYTE : BOOL
VAR_INPUT
	Destination : REFERENCE TO I_BYTE;
END_VAR
TryResolveAs_BYTE := _target.TryResolveAs_BYTE(Destination);
END_METHOD

METHOD PUBLIC TryResolveAs_DINT : BOOL
VAR_INPUT
	Destination : REFERENCE TO I_DINT;
END_VAR
TryResolveAs_DINT := _target.TryResolveAs_DINT(Destination);
END_METHOD

METHOD PUBLIC TryResolveAs_DT : BOOL
VAR_INPUT
	Destination : REFERENCE TO I_DT;
END_VAR
TryResolveAs_DT := _target.TryResolveAs_DT(Destination);
END_METHOD

METHOD PUBLIC TryResolveAs_DWORD : BOOL
VAR_INPUT
	Destination : REFERENCE TO I_DWORD;
END_VAR
TryResolveAs_DWORD := _target.TryResolveAs_DWORD(Destination);
END_METHOD

METHOD PUBLIC TryResolveAs_INT : BOOL
VAR_INPUT
	Destination : REFERENCE TO I_INT;
END_VAR
TryResolveAs_INT := _target.TryResolveAs_INT(Destination);
END_METHOD

METHOD PUBLIC TryResolveAs_LINT : BOOL
VAR_INPUT
	Destination : REFERENCE TO I_LINT;
END_VAR
TryResolveAs_LINT := _target.TryResolveAs_LINT(Destination);
END_METHOD

METHOD PUBLIC TryResolveAs_LREAL : BOOL
VAR_INPUT
	Destination : REFERENCE TO I_LREAL;
END_VAR
TryResolveAs_LREAL := _target.TryResolveAs_LREAL(Destination);
END_METHOD

METHOD PUBLIC TryResolveAs_LWORD : BOOL
VAR_INPUT
	Destination : REFERENCE TO I_LWORD;
END_VAR
TryResolveAs_LWORD := _target.TryResolveAs_LWORD(Destination);
END_METHOD

METHOD PUBLIC TryResolveAs_PVOID : BOOL
VAR_INPUT
	Destination : REFERENCE TO I_PVOID;
END_VAR
TryResolveAs_PVOID := _target.TryResolveAs_PVOID(Destination);
END_METHOD

METHOD PUBLIC TryResolveAs_REAL : BOOL
VAR_INPUT
	Destination : REFERENCE TO I_REAL;
END_VAR
TryResolveAs_REAL := _target.TryResolveAs_REAL(Destination);
END_METHOD

METHOD PUBLIC TryResolveAs_REFERENCE_TO : BOOL
VAR_INPUT
	Destination : REFERENCE TO I_REFERENCE_TO;
END_VAR
Destination := THIS^;
TryResolveAs_REFERENCE_TO := TRUE;
END_METHOD

METHOD PUBLIC TryResolveAs_SINT : BOOL
VAR_INPUT
	Destination : REFERENCE TO I_SINT;
END_VAR
TryResolveAs_SINT := _target.TryResolveAs_SINT(Destination);
END_METHOD

METHOD PUBLIC TryResolveAs_STRING : BOOL
VAR_INPUT
	Destination : REFERENCE TO I_STRING;
END_VAR
TryResolveAs_STRING := _target.TryResolveAs_STRING(Destination);
END_METHOD

METHOD PUBLIC TryResolveAs_TIME_OF_DAY : BOOL
VAR_INPUT
	Destination : REFERENCE TO I_TIME_OF_DAY;
END_VAR
TryResolveAs_TIME_OF_DAY := _target.TryResolveAs_TIME_OF_DAY(Destination);
END_METHOD

METHOD PUBLIC TryResolveAs_TOD : BOOL
VAR_INPUT
	Destination : REFERENCE TO I_TOD;
END_VAR
TryResolveAs_TOD := _target.TryResolveAs_TOD(Destination);
END_METHOD

METHOD PUBLIC TryResolveAs_UDINT : BOOL
VAR_INPUT
	Destination : REFERENCE TO I_UDINT;
END_VAR
TryResolveAs_UDINT := _target.TryResolveAs_UDINT(Destination);
END_METHOD

METHOD PUBLIC TryResolveAs_UINT : BOOL
VAR_INPUT
	Destination : REFERENCE TO I_UINT;
END_VAR
TryResolveAs_UINT := _target.TryResolveAs_UINT(Destination);
END_METHOD

METHOD PUBLIC TryResolveAs_ULINT : BOOL
VAR_INPUT
	Destination : REFERENCE TO I_ULINT;
END_VAR
TryResolveAs_ULINT := _target.TryResolveAs_ULINT(Destination);
END_METHOD

METHOD PUBLIC TryResolveAs_USINT : BOOL
VAR_INPUT
	Destination : REFERENCE TO I_USINT;
END_VAR
TryResolveAs_USINT := _target.TryResolveAs_USINT(Destination);
END_METHOD

METHOD PUBLIC TryResolveAs_WORD : BOOL
VAR_INPUT
	Destination : REFERENCE TO I_WORD;
END_VAR
TryResolveAs_WORD := _target.TryResolveAs_WORD(Destination);
END_METHOD

METHOD PUBLIC TryResolveAsAliasDatatype : BOOL
VAR_INPUT
	Destination : REFERENCE TO I_AliasDatatype;
END_VAR
TryResolveAsAliasDatatype := _target.TryResolveAsAliasDatatype(Destination);
END_METHOD

METHOD PUBLIC TryResolveAsArrayDatatype : BOOL
VAR_INPUT
	Destination : REFERENCE TO I_ArrayDatatype;
END_VAR
TryResolveAsArrayDatatype := _target.TryResolveAsArrayDatatype(Destination);
END_METHOD

METHOD PUBLIC TryResolveAsBitDatatype : BOOL
VAR_INPUT
	Destination : REFERENCE TO I_BIT;
END_VAR
TryResolveAsBitDatatype := _target.TryResolveAsBitDatatype(Destination);
END_METHOD

METHOD PUBLIC TryResolveAsEnumDatatype : BOOL
VAR_INPUT
	Destination : REFERENCE TO I_EnumDatatype;
END_VAR
TryResolveAsEnumDatatype := _target.TryResolveAsEnumDatatype(Destination);
END_METHOD

METHOD PUBLIC TryResolveAsInterfaceDatatype : BOOL
VAR_INPUT
	Destination : REFERENCE TO I_InterfaceDatatype;
END_VAR
TryResolveAsInterfaceDatatype := _target.TryResolveAsInterfaceDatatype(Destination);
END_METHOD

METHOD PUBLIC TryResolveAsStructuredDatatype : BOOL
VAR_INPUT
	Destination : REFERENCE TO I_StructuredDatatype;
END_VAR
TryResolveAsStructuredDatatype := _target.TryResolveAsStructuredDatatype(Destination);
END_METHOD

METHOD PUBLIC TryResolveAsUserDefinedDatatype : BOOL
VAR_INPUT
	Destination : REFERENCE TO I_UserDefinedDatatype;
END_VAR
TryResolveAsUserDefinedDatatype := _target.TryResolveAsUserDefinedDatatype(Destination);
END_METHOD

PROPERTY PUBLIC TypeName : T_MAXSTRING
GET
TypeName := concat('REFERENCE TO ', _target.TypeName);
END_GET
END_PROPERTY

END_FUNCTION_BLOCK

// ---- mobject-datatypes/Primitive/_NULL.TcPOU
{attribute 'linkalways'} 
{attribute 'no_explicit_call' := 'This FB is a CLASS and must be accessed using methods or properties'}
{attribute 'enable_dynamic_creation'}
FUNCTION_BLOCK _NULL EXTENDS DatatypeBase
VAR
END_VAR

PROPERTY PUBLIC Address : PVOID
GET
Address := 0;
END_GET
END_PROPERTY

METHOD PUBLIC ClearReference
VAR_INPUT
END_VAR
END_METHOD

METHOD PUBLIC Clone : I_Datatype
VAR
    pClone : POINTER TO _NULL;
END_VAR
pClone := __NEW(_NULL);
Clone := pClone^;
END_METHOD

PROPERTY PUBLIC IsNull : BOOL
GET
IsNull := TRUE;
END_GET
END_PROPERTY

METHOD PUBLIC SerializeWith
VAR_INPUT
	Serializer : I_Serializer;
END_VAR
Serializer.AddNull();
END_METHOD

PROPERTY PUBLIC Size : UDINT
GET
Size := 0;
END_GET
END_PROPERTY

METHOD TryDeserializeFrom : BOOL
VAR_INPUT
	Deserializer : I_Deserializer;
	Feedback : I_DeserializerFeedback;
END_VAR
END_METHOD

METHOD TryMakeReferenceTo : BOOL
VAR_INPUT
	Target : I_Datatype;
END_VAR
TryMakeReferenceTo := FALSE;
END_METHOD

PROPERTY PUBLIC TypeName : T_MAXSTRING
GET
TypeName := 'NULL';
END_GET
END_PROPERTY

END_FUNCTION_BLOCK

// ---- mobject-datatypes/Primitive/_BIT.TcPOU
{attribute 'linkalways'} 
{attribute 'no_explicit_call' := 'This FB is a CLASS and must be accessed using methods or properties'}
{attribute 'enable_dynamic_creation'}
FUNCTION_BLOCK _BIT EXTENDS DatatypeBase implements I_BIT
VAR
	initialised : BOOL;
	activeParent : I_StructuredDatatype;
	activeByteOffset : PVOID;
	activeBitOffset : DWORD;
END_VAR

PROPERTY PUBLIC Address : PVOID
GET
IF NOT initialised THEN 
	RETURN;
END_IF

Address := activeParent.Address + activeByteOffset;
END_GET
END_PROPERTY

PROPERTY PUBLIC BitOffset : DWORD
GET
IF NOT initialised THEN 
	RETURN;
END_IF

BitOffset := activeBitOffset;
END_GET
END_PROPERTY

PROPERTY PUBLIC ByteOffset : PVOID
GET
IF NOT initialised THEN 
	RETURN;
END_IF

ByteOffset := activeByteOffset;
END_GET
END_PROPERTY

METHOD PUBLIC ClearReference
VAR_INPUT
END_VAR
activeParent := 0;
activeByteOffset := 0;
activeBitOffset := 0;
initialised := FALSE;
END_METHOD

METHOD PUBLIC Clone : I_Datatype
VAR
    pClone : POINTER TO _BIT;
END_VAR
pClone := __NEW(_BIT);

IF initialised THEN
	pClone^.MakeReferenceTo(activeParent, activeByteOffset, activeBitOffset);
END_IF

Clone := pClone^;
END_METHOD

METHOD PRIVATE GetBitValue : BOOL
VAR
	pByte : POINTER TO BYTE := Address;
END_VAR
IF NOT initialised THEN
	RETURN;
END_IF

CASE activeBitOffset OF
	0: GetBitValue := pByte^.0;
	1: GetBitValue := pByte^.1;
	2: GetBitValue := pByte^.2;
	3: GetBitValue := pByte^.3;
	4: GetBitValue := pByte^.4;
	5: GetBitValue := pByte^.5;
	6: GetBitValue := pByte^.6;
	7: GetBitValue := pByte^.7;
END_CASE;
END_METHOD

METHOD PUBLIC MakeReferenceTo
VAR_INPUT
	Parent : I_StructuredDatatype;
	ByteOffset : PVOID;
	BitOffset : DWORD;
END_VAR
activeParent := Parent;
activeByteOffset := ByteOffset;
activeBitOffset := BitOffset AND 16#7;
initialised := TRUE;
END_METHOD

PROPERTY PUBLIC Parent : I_StructuredDatatype
GET
Parent := activeParent;
END_GET
END_PROPERTY

METHOD PUBLIC SerializeWith
VAR_INPUT
	Serializer : I_Serializer;
END_VAR
Serializer.AddBool(GetBitValue());
END_METHOD

METHOD PRIVATE SetBitValue : BOOL
VAR_INPUT
	Value : BOOL;
END_VAR
VAR
	pByte : POINTER TO BYTE := Address;
END_VAR
IF NOT initialised THEN
	RETURN;
END_IF

CASE activeBitOffset OF
	0: pByte^.0 := Value;
	1: pByte^.1 := Value;
	2: pByte^.2 := Value;
	3: pByte^.3 := Value;
	4: pByte^.4 := Value;
	5: pByte^.5 := Value;
	6: pByte^.6 := Value;
	7: pByte^.7 := Value;
END_CASE;
END_METHOD

PROPERTY PUBLIC Size : UDINT
GET
Size := 1;
END_GET
END_PROPERTY

METHOD PUBLIC TryConvertTo : BOOL
VAR_INPUT
	Destination : ANY;
END_VAR
TryConvertTo := TryConvert_BOOL_To_Destination(Value, Destination);
END_METHOD

METHOD PUBLIC TryConvertTo_ : BOOL
VAR_INPUT
	Destination : I_Datatype;
END_VAR
VAR
	resultofBitConversion : BOOL;
	destinationAs_BIT : I_BIT;
	destinationAs_BOOL : I_BOOL;
	destinationAs_BYTE : I_BYTE;
	destinationAs_DINT : I_DINT;
	destinationAs_DT : I_DT;
	destinationAs_DWORD : I_DWORD;
	destinationAs_INT : I_INT;
	destinationAs_LINT : I_LINT;
	destinationAs_LREAL : I_LREAL;
	destinationAs_LWORD : I_LWORD;
	destinationAs_REAL : I_REAL;
	destinationAs_SINT : I_SINT;
	destinationAs_STRING : I_STRING;
	destinationAs_TOD : I_TOD;
	destinationAs_UDINT : I_UDINT;
	destinationAs_UINT : I_UINT;
	destinationAs_ULINT : I_ULINT;
	destinationAs_USINT : I_USINT;
	destinationAs_WORD : I_WORD;
END_VAR
IF destination.TryResolveAs_BIT(destinationAs_BIT) AND_THEN TryConvert_BOOL_TO_BOOL(Value, resultofBitConversion) THEN
	destinationAs_BIT.Value := resultOfBitConversion;
	TryConvertTo_ := TRUE;
	RETURN;
END_IF

IF destination.TryResolveAs_BOOL(destinationAs_BOOL) THEN
	TryConvertTo_ := TryConvert_BOOL_TO_BOOL(Value, destinationAs_BOOL.Value);
	RETURN;
END_IF
		
IF destination.TryResolveAs_BYTE(destinationAs_BYTE) THEN
	TryConvertTo_ := TryConvert_BOOL_TO_BYTE(Value, destinationAs_BYTE.Value);
	RETURN;
END_IF

IF destination.TryResolveAs_DINT(destinationAs_DINT) THEN
	TryConvertTo_ := TryConvert_BOOL_TO_DINT(Value, destinationAs_DINT.Value);
	RETURN;
END_IF

IF destination.TryResolveAs_DT(destinationAs_DT) THEN
	TryConvertTo_ := TryConvert_BOOL_TO_DT(Value, destinationAs_DT.Value);
	RETURN;
END_IF

IF destination.TryResolveAs_DWORD(destinationAs_DWORD) THEN
	TryConvertTo_ := TryConvert_BOOL_TO_DWORD(Value, destinationAs_DWORD.Value);
	RETURN;
END_IF

IF destination.TryResolveAs_INT(destinationAs_INT) THEN
	TryConvertTo_ := TryConvert_BOOL_TO_INT(Value, destinationAs_INT.Value);
	RETURN;
END_IF

IF destination.TryResolveAs_LINT(destinationAs_LINT) THEN
	TryConvertTo_ := TryConvert_BOOL_TO_LINT(Value, destinationAs_LINT.Value);
	RETURN;
END_IF

IF destination.TryResolveAs_LREAL(destinationAs_LREAL) THEN
	TryConvertTo_ := TryConvert_BOOL_TO_LREAL(Value, destinationAs_LREAL.Value);
	RETURN;
END_IF

IF destination.TryResolveAs_LWORD(destinationAs_LWORD) THEN
	TryConvertTo_ := TryConvert_BOOL_TO_LWORD(Value, destinationAs_LWORD.Value);
	RETURN;
END_IF

IF destination.TryResolveAs_REAL(destinationAs_REAL) THEN
	TryConvertTo_ := TryConvert_BOOL_TO_REAL(Value, destinationAs_REAL.Value);
	RETURN;
END_IF

IF destination.TryResolveAs_SINT(destinationAs_SINT) THEN
	TryConvertTo_ := TryConvert_BOOL_TO_SINT(Value, destinationAs_SINT.Value);
	RETURN;
END_IF

IF destination.TryResolveAs_STRING(destinationAs_STRING) THEN
	TryConvertTo_ := TryConvert_BOOL_TO_STRING(Value, destinationAs_STRING.Value);
	RETURN;
END_IF

IF destination.TryResolveAs_TOD(destinationAs_TOD) THEN
	TryConvertTo_ := TryConvert_BOOL_TO_TOD(Value, destinationAs_TOD.Value);
	RETURN;
END_IF

IF destination.TryResolveAs_UDINT(destinationAs_UDINT) THEN
	TryConvertTo_ := TryConvert_BOOL_TO_UDINT(Value, destinationAs_UDINT.Value);
	RETURN;
END_IF

IF destination.TryResolveAs_UINT(destinationAs_UINT) THEN
	TryConvertTo_ := TryConvert_BOOL_TO_UINT(Value, destinationAs_UINT.Value);
	RETURN;
END_IF

IF destination.TryResolveAs_ULINT(destinationAs_ULINT) THEN
	TryConvertTo_ := TryConvert_BOOL_TO_ULINT(Value, destinationAs_ULINT.Value);
	RETURN;
END_IF

IF destination.TryResolveAs_USINT(destinationAs_USINT) THEN
	TryConvertTo_ := TryConvert_BOOL_TO_USINT(Value, destinationAs_USINT.Value);
	RETURN;
END_IF

IF destination.TryResolveAs_WORD(destinationAs_WORD) THEN
	TryConvertTo_ := TryConvert_BOOL_TO_WORD(Value, destinationAs_WORD.Value);
	RETURN;
END_IF
END_METHOD

METHOD TryDeserializeFrom : BOOL
VAR_INPUT
	Deserializer : I_Deserializer;
	Feedback : I_DeserializerFeedback;
END_VAR
VAR 
	value : BOOL;
END_VAR
IF NOT Deserializer.TryGetBool(value, Feedback) THEN
	RETURN;
END_IF

SetBitValue(value);
TryDeserializeFrom := TRUE;
END_METHOD

METHOD TryMakeReferenceTo : BOOL
VAR_INPUT
	Target : I_Datatype;
END_VAR
VAR
	targetAsBit : I_BIT;
END_VAR
IF NOT Target.Root.TryResolveAs_BIT(targetAsBit) THEN
	RETURN;
END_IF

MakeReferenceTo(targetAsBit.Parent, targetAsBit.ByteOffset, targetAsBit.BitOffset);
TryMakeReferenceTo := TRUE;
END_METHOD

METHOD PUBLIC TryResolveAs_BIT : BOOL
VAR_INPUT
	Destination : REFERENCE TO I_BIT;
END_VAR
Destination := THIS^;
TryResolveAs_BIT := TRUE;
END_METHOD

PROPERTY PUBLIC TypeName : T_MAXSTRING
GET
TypeName := 'BIT';
END_GET
END_PROPERTY

PROPERTY PUBLIC Value : BOOL
GET
Value := GetBitValue();
END_GET
SET
SetBitValue(Value);
END_SET
END_PROPERTY

END_FUNCTION_BLOCK

// ---- mobject-datatypes/Primitive/_ANY.TcPOU
{attribute 'linkalways'} 
{attribute 'no_explicit_call' := 'This FB is a CLASS and must be accessed using methods or properties'}
{attribute 'enable_dynamic_creation'}
FUNCTION_BLOCK _ANY EXTENDS Disposable IMPLEMENTS I_Any
VAR
	resolvedDatatype : I_Datatype;
END_VAR

METHOD PUBLIC Accept
VAR_INPUT
	Visitor : I_DatatypeVisitor;
END_VAR
IF resolvedDatatype = 0 THEN
	Visitor.VisitDatatype(THIS^);
	RETURN;
END_IF

Visitor.VisitDatatype(resolvedDatatype);
END_METHOD

PROPERTY PUBLIC Address : PVOID
GET
IF resolvedDatatype = 0 THEN
	RETURN;
END_IF

Address := resolvedDatatype.Address;
END_GET
END_PROPERTY

METHOD PUBLIC CanBecome : BOOL
VAR_INPUT
	Target : I_Datatype;
END_VAR
VAR
	targetAsAny : I_ANY;
END_VAR
IF Target.TryResolveAs_ANY(targetAsAny) THEN
	RETURN;
END_IF

CanBecome := TRUE;
END_METHOD

METHOD PUBLIC Clear
VAR_INPUT
END_VAR
ClearResolvedDatatype();
END_METHOD

METHOD PUBLIC ClearReference
VAR_INPUT
END_VAR
ClearResolvedDatatype();
END_METHOD

METHOD PRIVATE ClearResolvedDatatype
VAR_INPUT
END_VAR
VAR
	resolvedDatatypeAsAny : I_ANY;
END_VAR
IF resolvedDatatype = 0 THEN
	RETURN;
END_IF

IF resolvedDatatype.TryResolveAs_ANY(resolvedDatatypeAsAny) THEN
	resolvedDatatype := 0;
	RETURN;
END_IF

resolvedDatatype.Dispose();
resolvedDatatype := 0;
END_METHOD

METHOD PUBLIC Clone : I_Datatype
VAR
    pClone : POINTER TO _ANY;
END_VAR
IF resolvedDatatype = 0 THEN
	pClone := __NEW(_ANY);
	Clone := pClone^;
	RETURN;
END_IF

Clone := resolvedDatatype.Clone();
END_METHOD

METHOD PRIVATE CreateResolvedDatatype
VAR_INPUT
	DatatypeToClone : I_Datatype;
END_VAR
ClearResolvedDatatype();
resolvedDatatype := DatatypeToClone.Clone();
END_METHOD

METHOD FB_exit : BOOL
VAR_INPUT
	(* if TRUE, the exit method is called for exiting an instance that is copied afterwards (online change).*)
	bInCopyCode	: BOOL;
END_VAR
IF bInCopyCode THEN
	RETURN;
END_IF

ClearResolvedDatatype();
END_METHOD

METHOD PUBLIC IsEquivalentTo : BOOL
VAR_INPUT
	Datatype : I_Datatype;
END_VAR
IF resolvedDatatype = 0 THEN
	RETURN;
END_IF

IsEquivalentTo := resolvedDatatype.IsEquivalentTo(Datatype);
END_METHOD

PROPERTY PUBLIC IsNull : BOOL
GET
IF resolvedDatatype = 0 THEN
	RETURN;
END_IF

IsNull := resolvedDatatype.IsNull;
END_GET
END_PROPERTY

PROPERTY PUBLIC IsResolved : BOOL
GET
VAR
	resolvedDatatypeAsAny : I_ANY;
END_VAR
IF resolvedDatatype = 0 THEN
	RETURN;
END_IF

IF resolvedDatatype.TryResolveAs_ANY(resolvedDatatypeAsAny) THEN
	IsResolved := resolvedDatatypeAsAny.IsResolved;
	RETURN;
END_IF

IsResolved := TRUE;
END_GET
END_PROPERTY

PROPERTY PUBLIC IsUserDefined : BOOL
GET
IF resolvedDatatype = 0 THEN
	RETURN;
END_IF

IsUserDefined := resolvedDatatype.IsUserDefined;
END_GET
END_PROPERTY

PROPERTY PUBLIC Root : I_Datatype
GET
IF resolvedDatatype = 0 THEN
	Root := THIS^;
	RETURN;
END_IF

Root := resolvedDatatype.Root;
END_GET
END_PROPERTY

METHOD PUBLIC SerializeTypeWith
VAR_INPUT
	Serializer : I_Serializer;
END_VAR
Serializer.StartObject();
Serializer.AddKeyString('typeName',TypeName);
Serializer.EndObject();
END_METHOD

METHOD PUBLIC SerializeWith
VAR_INPUT
	Serializer : I_Serializer;
END_VAR
IF resolvedDatatype = 0 THEN
	RETURN;
END_IF

resolvedDatatype.SerializeWith(Serializer);
END_METHOD

PROPERTY PUBLIC Size : UDINT
GET
IF resolvedDatatype = 0 THEN
	RETURN;
END_IF

Size := resolvedDatatype.Size;
END_GET
END_PROPERTY

METHOD PUBLIC TryBecome : BOOL
VAR_INPUT
	Target : I_Datatype;
END_VAR
IF NOT CanBecome(Target) THEN
	RETURN;
END_IF

CreateResolvedDatatype(Target);
TryBecome := TRUE;
END_METHOD

METHOD PUBLIC TryConvertTo : BOOL
VAR_INPUT
	Destination : ANY;
END_VAR
IF resolvedDatatype = 0 THEN
	RETURN;
END_IF

TryConvertTo := resolvedDatatype.TryConvertTo(Destination);
END_METHOD

METHOD PUBLIC TryConvertTo_ : BOOL
VAR_INPUT
	Destination : I_Datatype;
END_VAR
IF resolvedDatatype = 0 THEN
	RETURN;
END_IF

TryConvertTo_ := resolvedDatatype.TryConvertTo_(Destination);
END_METHOD

METHOD PUBLIC TryCopyFrom : BOOL
VAR_INPUT
	Source : I_Datatype;
END_VAR
IF resolvedDatatype = 0 THEN
	RETURN;
END_IF

TryCopyFrom := resolvedDatatype.TryCopyFrom(Source);
END_METHOD

METHOD TryDeserializeFrom : BOOL
VAR_INPUT
	Deserializer : I_Deserializer;
	Feedback : I_DeserializerFeedback;
END_VAR
IF resolvedDatatype = 0 THEN
	RETURN;
END_IF

TryDeserializeFrom := resolvedDatatype.TryDeserializeFrom(Deserializer, Feedback);
END_METHOD

METHOD TryMakeReferenceTo : BOOL
VAR_INPUT
	Target : I_Datatype;
END_VAR
VAR
	targetAsAny : I_ANY;
END_VAR
IF Target.TryResolveAs_ANY(targetAsAny) THEN
	resolvedDatatype := Target;
	TryMakeReferenceTo := TRUE;
	RETURN;
END_IF

CreateResolvedDatatype(Target);
TryMakeReferenceTo := resolvedDatatype.TryMakeReferenceTo(Target);
END_METHOD

METHOD PUBLIC TryResolveAs_ANY : BOOL
VAR_INPUT
	Destination : REFERENCE TO I_ANY;
END_VAR
Destination := THIS^;
TryResolveAs_ANY := TRUE;
END_METHOD

METHOD PUBLIC TryResolveAs_BIT : BOOL
VAR_INPUT
	Destination : REFERENCE TO I_BIT;
END_VAR
IF resolvedDatatype = 0 THEN
	RETURN;
END_IF

TryResolveAs_BIT := resolvedDatatype.TryResolveAs_BIT(Destination);
END_METHOD

METHOD PUBLIC TryResolveAs_BOOL : BOOL
VAR_INPUT
	Destination : REFERENCE TO I_BOOL;
END_VAR
IF resolvedDatatype = 0 THEN
	RETURN;
END_IF

TryResolveAs_BOOL := resolvedDatatype.TryResolveAs_BOOL(Destination);
END_METHOD

METHOD PUBLIC TryResolveAs_BYTE : BOOL
VAR_INPUT
	Destination : REFERENCE TO I_BYTE;
END_VAR
IF resolvedDatatype = 0 THEN
	RETURN;
END_IF

TryResolveAs_BYTE := resolvedDatatype.TryResolveAs_BYTE(Destination);
END_METHOD

METHOD PUBLIC TryResolveAs_DINT : BOOL
VAR_INPUT
	Destination : REFERENCE TO I_DINT;
END_VAR
IF resolvedDatatype = 0 THEN
	RETURN;
END_IF

TryResolveAs_DINT := resolvedDatatype.TryResolveAs_DINT(Destination);
END_METHOD

METHOD PUBLIC TryResolveAs_DT : BOOL
VAR_INPUT
	Destination : REFERENCE TO I_DT;
END_VAR
IF resolvedDatatype = 0 THEN
	RETURN;
END_IF

TryResolveAs_DT := resolvedDatatype.TryResolveAs_DT(Destination);
END_METHOD

METHOD PUBLIC TryResolveAs_DWORD : BOOL
VAR_INPUT
	Destination : REFERENCE TO I_DWORD;
END_VAR
IF resolvedDatatype = 0 THEN
	RETURN;
END_IF

TryResolveAs_DWORD := resolvedDatatype.TryResolveAs_DWORD(Destination);
END_METHOD

METHOD PUBLIC TryResolveAs_INT : BOOL
VAR_INPUT
	Destination : REFERENCE TO I_INT;
END_VAR
IF resolvedDatatype = 0 THEN
	RETURN;
END_IF

TryResolveAs_INT := resolvedDatatype.TryResolveAs_INT(Destination);
END_METHOD

METHOD PUBLIC TryResolveAs_LINT : BOOL
VAR_INPUT
	Destination : REFERENCE TO I_LINT;
END_VAR
IF resolvedDatatype = 0 THEN
	RETURN;
END_IF

TryResolveAs_LINT := resolvedDatatype.TryResolveAs_LINT(Destination);
END_METHOD

METHOD PUBLIC TryResolveAs_LREAL : BOOL
VAR_INPUT
	Destination : REFERENCE TO I_LREAL;
END_VAR
IF resolvedDatatype = 0 THEN
	RETURN;
END_IF

TryResolveAs_LREAL := resolvedDatatype.TryResolveAs_LREAL(Destination);
END_METHOD

METHOD PUBLIC TryResolveAs_LWORD : BOOL
VAR_INPUT
	Destination : REFERENCE TO I_LWORD;
END_VAR
IF resolvedDatatype = 0 THEN
	RETURN;
END_IF

TryResolveAs_LWORD := resolvedDatatype.TryResolveAs_LWORD(Destination);
END_METHOD

METHOD PUBLIC TryResolveAs_PVOID : BOOL
VAR_INPUT
	Destination : REFERENCE TO I_PVOID;
END_VAR
IF resolvedDatatype = 0 THEN
	RETURN;
END_IF

TryResolveAs_PVOID := resolvedDatatype.TryResolveAs_PVOID(Destination);
END_METHOD

METHOD PUBLIC TryResolveAs_REAL : BOOL
VAR_INPUT
	Destination : REFERENCE TO I_REAL;
END_VAR
IF resolvedDatatype = 0 THEN
	RETURN;
END_IF

TryResolveAs_REAL := resolvedDatatype.TryResolveAs_REAL(Destination);
END_METHOD

METHOD PUBLIC TryResolveAs_REFERENCE_TO : BOOL
VAR_INPUT
	Destination : REFERENCE TO I_REFERENCE_TO;
END_VAR
IF resolvedDatatype = 0 THEN
	RETURN;
END_IF

TryResolveAs_REFERENCE_TO := resolvedDatatype.TryResolveAs_REFERENCE_TO(Destination);
END_METHOD

METHOD PUBLIC TryResolveAs_SINT : BOOL
VAR_INPUT
	Destination : REFERENCE TO I_SINT;
END_VAR
IF resolvedDatatype = 0 THEN
	RETURN;
END_IF

TryResolveAs_SINT := resolvedDatatype.TryResolveAs_SINT(Destination);
END_METHOD

METHOD PUBLIC TryResolveAs_STRING : BOOL
VAR_INPUT
	Destination : REFERENCE TO I_STRING;
END_VAR
IF resolvedDatatype = 0 THEN
	RETURN;
END_IF

TryResolveAs_STRING := resolvedDatatype.TryResolveAs_STRING(Destination);
END_METHOD

METHOD PUBLIC TryResolveAs_TIME_OF_DAY : BOOL
VAR_INPUT
	Destination : REFERENCE TO I_TIME_OF_DAY;
END_VAR
IF resolvedDatatype = 0 THEN
	RETURN;
END_IF

TryResolveAs_TIME_OF_DAY := resolvedDatatype.TryResolveAs_TIME_OF_DAY(Destination);
END_METHOD

METHOD PUBLIC TryResolveAs_TOD : BOOL
VAR_INPUT
	Destination : REFERENCE TO I_TOD;
END_VAR
IF resolvedDatatype = 0 THEN
	RETURN;
END_IF

TryResolveAs_TOD := resolvedDatatype.TryResolveAs_TOD(Destination);
END_METHOD

METHOD PUBLIC TryResolveAs_UDINT : BOOL
VAR_INPUT
	Destination : REFERENCE TO I_UDINT;
END_VAR
IF resolvedDatatype = 0 THEN
	RETURN;
END_IF

TryResolveAs_UDINT := resolvedDatatype.TryResolveAs_UDINT(Destination);
END_METHOD

METHOD PUBLIC TryResolveAs_UINT : BOOL
VAR_INPUT
	Destination : REFERENCE TO I_UINT;
END_VAR
IF resolvedDatatype = 0 THEN
	RETURN;
END_IF

TryResolveAs_UINT := resolvedDatatype.TryResolveAs_UINT(Destination);
END_METHOD

METHOD PUBLIC TryResolveAs_ULINT : BOOL
VAR_INPUT
	Destination : REFERENCE TO I_ULINT;
END_VAR
IF resolvedDatatype = 0 THEN
	RETURN;
END_IF

TryResolveAs_ULINT := resolvedDatatype.TryResolveAs_ULINT(Destination);
END_METHOD

METHOD PUBLIC TryResolveAs_USINT : BOOL
VAR_INPUT
	Destination : REFERENCE TO I_USINT;
END_VAR
IF resolvedDatatype = 0 THEN
	RETURN;
END_IF

TryResolveAs_USINT := resolvedDatatype.TryResolveAs_USINT(Destination);
END_METHOD

METHOD PUBLIC TryResolveAs_WORD : BOOL
VAR_INPUT
	Destination : REFERENCE TO I_WORD;
END_VAR
IF resolvedDatatype = 0 THEN
	RETURN;
END_IF

TryResolveAs_WORD := resolvedDatatype.TryResolveAs_WORD(Destination);
END_METHOD

METHOD PUBLIC TryResolveAsAliasDatatype : BOOL
VAR_INPUT
	Destination : REFERENCE TO I_AliasDatatype;
END_VAR
IF resolvedDatatype = 0 THEN
	RETURN;
END_IF

TryResolveAsAliasDatatype := resolvedDatatype.TryResolveAsAliasDatatype(Destination);
END_METHOD

METHOD PUBLIC TryResolveAsArrayDatatype : BOOL
VAR_INPUT
	Destination : REFERENCE TO I_ArrayDatatype;
END_VAR
IF resolvedDatatype = 0 THEN
	RETURN;
END_IF

TryResolveAsArrayDatatype := resolvedDatatype.TryResolveAsArrayDatatype(Destination);
END_METHOD

METHOD PUBLIC TryResolveAsBitDatatype : BOOL
VAR_INPUT
	Destination : REFERENCE TO I_BIT;
END_VAR
IF resolvedDatatype = 0 THEN
	RETURN;
END_IF

TryResolveAsBitDatatype := resolvedDatatype.TryResolveAsBitDatatype(Destination);
END_METHOD

METHOD PUBLIC TryResolveAsEnumDatatype : BOOL
VAR_INPUT
	Destination : REFERENCE TO I_EnumDatatype;
END_VAR
IF resolvedDatatype = 0 THEN
	RETURN;
END_IF

TryResolveAsEnumDatatype := resolvedDatatype.TryResolveAsEnumDatatype(Destination);
END_METHOD

METHOD PUBLIC TryResolveAsInterfaceDatatype : BOOL
VAR_INPUT
	Destination : REFERENCE TO I_InterfaceDatatype;
END_VAR
IF resolvedDatatype = 0 THEN
	RETURN;
END_IF

TryResolveAsInterfaceDatatype := resolvedDatatype.TryResolveAsInterfaceDatatype(Destination);
END_METHOD

METHOD PUBLIC TryResolveAsStructuredDatatype : BOOL
VAR_INPUT
	Destination : REFERENCE TO I_StructuredDatatype;
END_VAR
IF resolvedDatatype = 0 THEN
	RETURN;
END_IF

TryResolveAsStructuredDatatype := resolvedDatatype.TryResolveAsStructuredDatatype(Destination);
END_METHOD

METHOD PUBLIC TryResolveAsUserDefinedDatatype : BOOL
VAR_INPUT
	Destination : REFERENCE TO I_UserDefinedDatatype;
END_VAR
IF resolvedDatatype = 0 THEN
	RETURN;
END_IF

TryResolveAsUserDefinedDatatype := resolvedDatatype.TryResolveAsUserDefinedDatatype(Destination);
END_METHOD

PROPERTY PUBLIC TypeName : T_MAXSTRING
GET
IF resolvedDatatype = 0 THEN
	TypeName := 'ANY';
	RETURN;
END_IF

TypeName := resolvedDatatype.TypeName;
END_GET
END_PROPERTY

END_FUNCTION_BLOCK

// ---- mobject-datatypes/Primitive/_TIME_OF_DAY.TcPOU
{attribute 'linkalways'} 
{attribute 'no_explicit_call' := 'This FB is a CLASS and must be accessed using methods or properties'}
{attribute 'enable_dynamic_creation'}
FUNCTION_BLOCK _TIME_OF_DAY EXTENDS DatatypeBase IMPLEMENTS I_TIME_OF_DAY
VAR
	localData : TIME_OF_DAY;
	activeData : REFERENCE TO TIME_OF_DAY REF= localData;
END_VAR

PROPERTY PUBLIC Address : PVOID
GET
Address := ADR(activeData);
END_GET
END_PROPERTY

METHOD PUBLIC ClearReference
VAR_INPUT
END_VAR
activeData REF= localData;
END_METHOD

METHOD PUBLIC Clone : I_Datatype
VAR
    pClone : POINTER TO _TIME_OF_DAY;
END_VAR
pClone := __NEW(_TIME_OF_DAY(InitialValue := Value));
Clone := pClone^;
END_METHOD

METHOD FB_init : BOOL
VAR_INPUT
	bInitRetains : BOOL; // if TRUE, the retain variables are initialized (warm start / cold start)
	bInCopyCode : BOOL;  // if TRUE, the instance afterwards gets moved WORDo the copy code (online change)
	InitialValue : TIME_OF_DAY;
END_VAR
localData := InitialValue;
END_METHOD

METHOD PUBLIC MakeReferenceTo
VAR_INPUT
	ReferenceTarget : REFERENCE TO TIME_OF_DAY;
END_VAR
activeData REF= ReferenceTarget;
END_METHOD

METHOD PUBLIC SerializeWith
VAR_INPUT
	Serializer : I_Serializer;
END_VAR
Serializer.AddTod(activeData);
END_METHOD

PROPERTY PUBLIC Size : UDINT
GET
Size := SIZEOF(activeData);
END_GET
END_PROPERTY

METHOD TryDeserializeFrom : BOOL
VAR_INPUT
	Deserializer : I_Deserializer;
	Feedback : I_DeserializerFeedback;
END_VAR
TryDeserializeFrom := Deserializer.TryGetTod(activeData, Feedback);
END_METHOD

METHOD TryMakeReferenceTo : BOOL
VAR_INPUT
	Target : I_Datatype;
END_VAR
VAR
	pTargetData : POINTER TO TIME_OF_DAY;
END_VAR
IF NOT IsEquivalentTo(Target) THEN
	RETURN;
END_IF

pTargetData := Target.Address;
activeData REF= pTargetData^;
TryMakeReferenceTo := TRUE;
END_METHOD

METHOD PUBLIC TryResolveAs_TIME_OF_DAY : BOOL
VAR_INPUT
	Destination : REFERENCE TO I_TIME_OF_DAY;
END_VAR
Destination := THIS^;
TryResolveAs_TIME_OF_DAY := TRUE;
END_METHOD

PROPERTY PUBLIC TypeName : T_MAXSTRING
GET
TypeName := 'TIME_OF_DAY';
END_GET
END_PROPERTY

{warning disable C5410}
PROPERTY PUBLIC Value : REFERENCE TO TIME_OF_DAY
{warning restore C5410}
GET
Value REF= activeData;
END_GET
END_PROPERTY

END_FUNCTION_BLOCK

// ---- mobject-datatypes/Primitive/_PVOID.TcPOU
{attribute 'linkalways'} 
{attribute 'no_explicit_call' := 'This FB is a CLASS and must be accessed using methods or properties'}
{attribute 'enable_dynamic_creation'}
FUNCTION_BLOCK _PVOID EXTENDS DatatypeBase IMPLEMENTS I_PVOID
VAR
	localData : PVOID;
	activeData : REFERENCE TO PVOID REF= localData;
END_VAR

PROPERTY PUBLIC Address : PVOID
GET
Address := ADR(activeData);
END_GET
END_PROPERTY

METHOD PUBLIC ClearReference
VAR_INPUT
END_VAR
activeData REF= localData;
END_METHOD

METHOD PUBLIC Clone : I_Datatype
VAR
    pClone : POINTER TO _PVOID;
END_VAR
pClone := __NEW(_PVOID);
Clone := pClone^;
END_METHOD

METHOD PUBLIC MakeReferenceTo
VAR_INPUT
	ReferenceTarget : REFERENCE TO PVOID;
END_VAR
activeData REF= ReferenceTarget;
END_METHOD

METHOD PUBLIC SerializeWith
VAR_INPUT
	Serializer : I_Serializer;
END_VAR
VAR
	pVoidAsString : T_MAXSTRING;
END_VAR
pVoidAsString := pvoid_To_string(activeData);
Serializer.AddString(pVoidAsString);
END_METHOD

PROPERTY PUBLIC Size : UDINT
GET
Size := SIZEOF(activeData);
END_GET
END_PROPERTY

METHOD TryDeserializeFrom : BOOL
VAR_INPUT
	Deserializer : I_Deserializer;
	Feedback : I_DeserializerFeedback;
END_VAR
VAR
	pVoidAsString : T_MAXSTRING;
END_VAR
IF NOT Deserializer.TryGetString(pVoidAsString, Feedback) THEN
	RETURN;
END_IF

activeData := STRING_TO_PVOID(pVoidAsString);
TryDeserializeFrom := TRUE;
END_METHOD

METHOD TryMakeReferenceTo : BOOL
VAR_INPUT
	Target : I_Datatype;
END_VAR
VAR
	pTargetData : POINTER TO PVOID;
END_VAR
IF NOT IsEquivalentTo(Target) THEN
	RETURN;
END_IF

pTargetData := Target.Address;
activeData REF= pTargetData^;
TryMakeReferenceTo := TRUE;
END_METHOD

METHOD PUBLIC TryResolveAs_PVOID : BOOL
VAR_INPUT
	Destination : REFERENCE TO I_PVOID;
END_VAR
Destination := THIS^;
TryResolveAs_PVOID := TRUE;
END_METHOD

PROPERTY PUBLIC TypeName : T_MAXSTRING
GET
TypeName := 'PVOID';
END_GET
END_PROPERTY

{warning disable C5410}
PROPERTY PUBLIC Value : REFERENCE TO PVOID
{warning restore C5410}
GET
Value REF= activeData;
END_GET
END_PROPERTY

END_FUNCTION_BLOCK

// ---- mobject-datatypes/_Internal/Datatype/AliasDatatypeBase.TcPOU
{attribute 'linkalways'} 
{attribute 'no_explicit_call' := 'This FB is a CLASS and must be accessed using methods or properties'}
{attribute 'enable_dynamic_creation'}
FUNCTION_BLOCK ABSTRACT AliasDatatypeBase EXTENDS UserDefinedDatatypeBase IMPLEMENTS I_AliasDatatype
VAR
	_baseDatatype : I_Datatype; // this value is the single level down
END_VAR

METHOD PROTECTED AddBaseDatatype
VAR_INPUT
	BaseType : I_Datatype;
END_VAR
_baseDatatype := BaseType;
END_METHOD

PROPERTY PUBLIC BaseDatatype : I_Datatype
GET
BaseDatatype := _baseDatatype;
END_GET
END_PROPERTY

METHOD PUBLIC IsEquivalentTo : BOOL
VAR_INPUT
	Datatype : I_Datatype;
END_VAR
// overrides as alias are always wrapped up, so it should defer to it's root
IsEquivalentTo := Root.IsEquivalentTo(Datatype.Root);
END_METHOD

METHOD PROTECTED OnSerializeTypeWith
VAR_INPUT
	Serializer : I_Serializer;
END_VAR
SUPER^.OnSerializeTypeWith(Serializer);
Serializer.AddKey('baseDatatype');
_baseDatatype.SerializeTypeWith(Serializer);
END_METHOD

PROPERTY PUBLIC Root : I_Datatype
GET
Root := _baseDatatype.Root;
END_GET
END_PROPERTY

METHOD PUBLIC SerializeWith
VAR_INPUT
	Serializer : I_Serializer;
END_VAR
_baseDatatype.SerializeWith(Serializer);
END_METHOD

METHOD PUBLIC TryConvertTo : BOOL
VAR_INPUT
	Destination : ANY;
END_VAR
TryConvertTo := _baseDatatype.TryConvertTo(Destination);
END_METHOD

METHOD PUBLIC TryConvertTo_ : BOOL
VAR_INPUT
	Destination : I_Datatype;
END_VAR
TryConvertTo_ := _baseDatatype.TryConvertTo_(Destination);
END_METHOD

METHOD TryDeserializeFrom : BOOL
VAR_INPUT
	Deserializer : I_Deserializer;
	Feedback : I_DeserializerFeedback;
END_VAR
TryDeserializeFrom := _baseDatatype.TryDeserializeFrom(Deserializer, Feedback);
END_METHOD

METHOD PUBLIC TryResolveAsAliasDatatype : BOOL
VAR_INPUT
	Destination : REFERENCE TO I_AliasDatatype;
END_VAR
Destination := THIS^;
TryResolveAsAliasDatatype := TRUE;
END_METHOD

PROPERTY PUBLIC TypeName : T_MAXSTRING
GET
TypeName := 'ALIAS';
END_GET
END_PROPERTY

END_FUNCTION_BLOCK

// ---- mobject-datatypes/_Internal/Datatype/UserDefinedDatatypeBase.TcPOU
{attribute 'linkalways'} 
{attribute 'no_explicit_call' := 'This FB is a CLASS and must be accessed using methods or properties'}
{attribute 'enable_dynamic_creation'}
FUNCTION_BLOCK ABSTRACT UserDefinedDatatypeBase EXTENDS DatatypeBase IMPLEMENTS I_UserDefinedDatatype
VAR
END_VAR

PROPERTY PUBLIC ABSTRACT Identifier : T_MAXSTRING
GET
END_GET
END_PROPERTY

METHOD PUBLIC IsEquivalentTo : BOOL
VAR_INPUT
	Datatype : I_Datatype;
END_VAR
VAR
	datatypeAsUdt : I_UserDefinedDatatype;
END_VAR
IF NOT Datatype.Root.TryResolveAsUserDefinedDatatype(datatypeAsUdt) THEN
	RETURN;
END_IF

IF datatypeAsUdt.Identifier <> Identifier THEN
	RETURN;
END_IF

IsEquivalentTo := SUPER^.IsEquivalentTo(Datatype);
END_METHOD

PROPERTY PUBLIC IsUserDefined : BOOL
GET
IsUserDefined := TRUE;
END_GET
END_PROPERTY

METHOD PROTECTED OnSerializeTypeWith
VAR_INPUT
	Serializer : I_Serializer;
END_VAR
SUPER^.OnSerializeTypeWith(Serializer);
Serializer.AddKeyString('identifier',Identifier);
END_METHOD

METHOD PUBLIC TryCopyFrom : BOOL
VAR_INPUT
	Source : I_Datatype;
END_VAR
VAR
	sourceAsUdt : I_UserDefinedDatatype;
END_VAR
IF NOT Source.TryResolveAsUserDefinedDatatype(sourceAsUdt) THEN
	RETURN;
END_IF

IF sourceAsUdt.Identifier <> Identifier THEN
	RETURN;
END_IF

TryCopyFrom := SUPER^.TryCopyFrom(Source);
END_METHOD

METHOD PUBLIC TryResolveAsUserDefinedDatatype : BOOL
VAR_INPUT
	Destination : REFERENCE TO I_UserDefinedDatatype;
END_VAR
Destination := THIS^;
TryResolveAsUserDefinedDatatype := TRUE;
END_METHOD

END_FUNCTION_BLOCK

// ---- mobject-datatypes/_Internal/Datatype/ArrayDatatypeBase_3D.TcPOU
{attribute 'linkalways'} 
{attribute 'no_explicit_call' := 'This FB is a CLASS and must be accessed using methods or properties'}
{attribute 'enable_dynamic_creation'}
FUNCTION_BLOCK ABSTRACT ArrayDatatypeBase_3D EXTENDS UserDefinedDatatypeBase IMPLEMENTS I_ArrayDatatype_3D
VAR
END_VAR

PROPERTY PUBLIC ABSTRACT BaseDatatype : I_Datatype
GET
END_GET
END_PROPERTY

PROPERTY Dimention : UDINT
GET
Dimention := 3;
END_GET
END_PROPERTY

